// TIA Portal V20 export
// export: Created 2025-12-01T14:56:53.2273381Z, ExportSetting None, DisplayName Totally Integrated Automation Portal, DisplayVersion V20 Update 3, DisplayName TIA Portal Openness, DisplayVersion V20 Update 3, DisplayName TIA Portal Version Control Interface, DisplayVersion V20 Update 3, DisplayName STEP 7 Professional, DisplayVersion V20 Update 3, DisplayName STEP 7 Safety, DisplayVersion V20 Update 2, DisplayName WinCC Basic/Comfort/Advanced, DisplayVersion V20 Update 3, DisplayName WinCC Professional, DisplayVersion V20 Update 3, DisplayName WinCC Unified, DisplayVersion V20 Update 3
FUNCTION_BLOCK "FB368_DesapilCubetas_ERAMAN"   // FB368, LAD
{ S7_Optimized_Access := 'FALSE' }
AUTHOR : PASO
NAME : 20160509
VERSION : 3.8
// stored: AutoNumber false, SetENOAutomatically false
   VAR_INPUT
      Mesa : UInt;   // Mesa de la FB
      Error_Tx : Bool;   // Error en el Tx
      EnTension : Bool;   // Existe Tension en la Mesa
      Termico_Tx : Bool;   // Termico motorrodillo
      PhsMx : Bool;   // Presencia en mesa
      Phs_Pos_Desapil : Bool;   // Posición cilindro medio
      Phs_en_Pinza : Bool;   // Presencia en pinza
      Avance_Tx : Bool;   // Avance del Tx
      CL_UP : Bool;   // Posición cilindro arriba
      CL_DW : Bool;   // Posición cilindro abajo
      EnMovimiento_CL : Bool;
      Gripper_Open : Bool;   // Posición pinza abierta
      Gripper_Close : Bool;   // Posición pinza cerrada
      EnMovimiento_Gripper : Bool;
      TP_UP : Bool;   // Posición tope arriba
      TP_DW : Bool;   // Posición tope abajo
      EnMovimiento_TP : Bool;   // En movimiento el TP1
      MAnt_DescargaAct : Bool;   // E1 >> Mesa Anterior DescargaAct
      AVTF_MAnt_Mx : Bool;
      PTF_Mx_MSig : Bool;
      FTF_Mx_MSig : Bool;
      V_CNT_pHsMx : Int := 1000;   // Valor de Presencia
      V_CNTSeg_pHsMx : Int := 2000;
      V_CNT_ApHsMx : Int := 500;
      V_CNTSeg_ApHsMx : Int := 2000;
      V_CNT_Simultaneo : Int := 2000;   // Valor de Simultaneo
      V_InicioSimultaneo : Int := 0;   // Inicio de Simultaneo. Nota: <= V_CNT_Simultaneo
      V_FinSimultaneo : Int := 0;   // Final de Simultaneo. Nota: <= V_InicioSimultaneo
      V_GripperAbrir : Time := T#200ms;
      V_TOut_Tx_Mx : Int := 10000;   // TimeOut de Entrada por E1
      V_TOut_TP : Int := 2000;   // TimeOut de Tope
      V_TOut_Apil_UPDW : Int := 5000;
      V_TOut_Gripper : Int := 2000;
   END_VAR
   VAR_OUTPUT
      AVTF_Mx_MSig : Bool;
      PTF_MAnt_Mx : Bool;   // E1 >> Mesa Anterior PTF
      FTF_MAnt_Mx : Bool;   // E1 >> Mesa Anterior FTF
      P_Mens_Mx_MSig : Bool;   // S3 >> Mesa Siguiente P_Mens
   END_VAR
   VAR
      Mx_ET00 : Bool;
      Mx_ET01 : Bool;
      Mx_ET02 : Bool;
      Mx_ET08 : Bool;
      Mx_ET09 : Bool;
      Mx_ET10 : Bool;
      Mx_ET11 : Bool;
      Mx_ET12 : Bool;
      Mx_ET50 : Bool;
      Mx_ET51 : Bool;
      Mx_ET501 : Bool;
      Mx_ET502 : Bool;
      Mx_ET503 : Bool;
      Mx_ET504 : Bool;
      Mx_ET505 : Bool;
      Mx_ET506 : Bool;
      STAT_AVTF_Mx_MSig { S7_SetPoint := 'True'} : Bool;
      STAT_FTF_MAnt_Mx : Bool;   // Interna >> FTF de MAnt >> Mx
      MA_Subir_CL : Bool;   // Salida para subir cilindro
      MA_Bajar_CL : Bool;   // Salida para bajar cilindro
      MA_Gripper_Cerrar : Bool;   // Salida cerrar gripper
      MA_Gripper_Abrir : Bool;   // Salida abrir gripper
      En_Movimiento : Bool;
      Simultaneo_Mx : Bool;   // Activo Simultaneo E1
      TMP_Gripper_Cerrar { S7_SetPoint := 'True'} : TON_TIME;
      CNT_pHsMx { S7_SetPoint := 'True'} : "FB910_CNT_UHS";   // CNT de la Presencia
      CNTSeg_pHsMx { S7_SetPoint := 'True'} : "FB910_CNT_UHS";   // CNT de Seguridad de la Presencia
      CNT_ApHsMx { S7_SetPoint := 'True'} : "FB910_CNT_UHS";   // CNT de la Ausencia
      CNTSeg_ApHsMx { S7_SetPoint := 'True'} : "FB910_CNT_UHS";   // CNT de Seguridad de la Ausencia
      CNT_Simultaneo { S7_SetPoint := 'True'} : "FB910_CNT_UHS";   // CNT de Simultaneo
      TMP_EnTension { S7_SetPoint := 'True'} : "FB910_CNT_UHS";
      TOut_Av { S7_SetPoint := 'True'} : "FB910_CNT_UHS";
      TOut_UPDW { S7_SetPoint := 'True'} : "FB910_CNT_UHS";
      TOut_Gripper { S7_SetPoint := 'True'} : "FB910_CNT_UHS";
      TOut_Subir_TP { S7_SetPoint := 'True'} : "FB910_CNT_UHS";
      TOut_Bajar_TP { S7_SetPoint := 'True'} : "FB910_CNT_UHS";
      Manual : "MoviManualMesa_Eraman";
   END_VAR
   VAR_TEMP
      EstadoZona : "EstadoZona";   // Estado de Zona de la Mesa
      EstadoVI : "EstadosMesa_ERAMAN";   // Estado del Vehiculo Inteliguente de la Mesa
      EstadoMaquina : "EstadoMaquina";
      ConfigFB : "UDT_ConfigFB";   // Configuracion de la FB de la Mesa
      Aux_ET00 : Bool;
   END_VAR
BEGIN

REGION Network 1: INICIALIZAR - Recoger las Variables de Estado de la Mesa
   // Se recoge - Estado_CBx
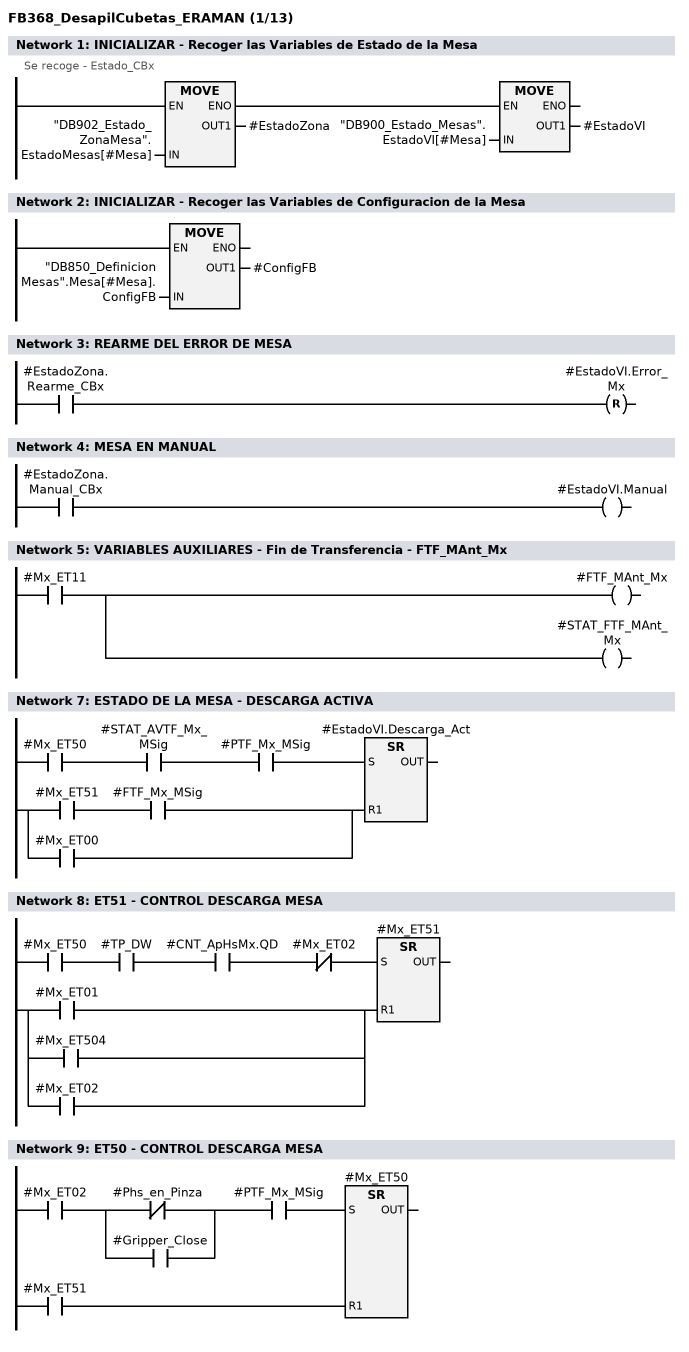
   RUNG wire#powerrail
      Move(in := "DB902_Estado_ZonaMesa".EstadoMesas[#Mesa], out1 => #EstadoZona)
      Move(in := "DB900_Estado_Mesas".EstadoVI[#Mesa], out1 => #EstadoVI)
   END_RUNG
   // the same network as SCL:
   #EstadoZona := "DB902_Estado_ZonaMesa".EstadoMesas[#Mesa];
   #EstadoVI := "DB900_Estado_Mesas".EstadoVI[#Mesa];
END_REGION

REGION Network 2: INICIALIZAR - Recoger las Variables de Configuracion de la Mesa
   RUNG wire#powerrail
      Move(in := "DB850_DefinicionMesas".Mesa[#Mesa].ConfigFB, out1 => #ConfigFB)
   END_RUNG
   // the same network as SCL:
   #ConfigFB := "DB850_DefinicionMesas".Mesa[#Mesa].ConfigFB;
END_REGION

REGION Network 3: REARME DEL ERROR DE MESA
   RUNG wire#powerrail
      Contact( #EstadoZona.Rearme_CBx )
      R_Coil( #EstadoVI.Error_Mx )
   END_RUNG
   // the same network as SCL:
   IF #EstadoZona.Rearme_CBx THEN #EstadoVI.Error_Mx := FALSE; END_IF;
END_REGION

REGION Network 4: MESA EN MANUAL
   RUNG wire#powerrail
      Contact( #EstadoZona.Manual_CBx )
      Coil( #EstadoVI.Manual )
   END_RUNG
   // the same network as SCL:
   #EstadoVI.Manual := #EstadoZona.Manual_CBx;
END_REGION

REGION Network 5: VARIABLES AUXILIARES - Fin de Transferencia - FTF_MAnt_Mx
   RUNG wire#powerrail
      Contact( #Mx_ET11 )
      wire#w1
      Coil( #FTF_MAnt_Mx )
   END_RUNG
   RUNG wire#w1
      Coil( #STAT_FTF_MAnt_Mx )
   END_RUNG
   // the same network as SCL:
   #FTF_MAnt_Mx := #Mx_ET11;
   #STAT_FTF_MAnt_Mx := #Mx_ET11;
END_REGION

REGION Network 6: ----------------------GRAFCET DESCARGA---------------------------
END_REGION

REGION Network 7: ESTADO DE LA MESA - DESCARGA ACTIVA
   RUNG wire#powerrail
      Contact( #Mx_ET50 )
      Contact( #STAT_AVTF_Mx_MSig )
      Contact( #PTF_Mx_MSig )
      S_SR(operand := #EstadoVI.Descarga_Act, r1 := wire#w1)
   END_RUNG
   RUNG wire#powerrail
      Contact( #Mx_ET51 )
      Contact( #FTF_Mx_MSig )
   END_RUNG wire#w1
   RUNG wire#powerrail
      Contact( #Mx_ET00 )
   END_RUNG wire#w1
   // the same network as SCL:
   IF #Mx_ET50 AND #STAT_AVTF_Mx_MSig AND #PTF_Mx_MSig THEN
       #EstadoVI.Descarga_Act := TRUE;   // SR flip-flop
   END_IF;
   IF (#Mx_ET51 AND #FTF_Mx_MSig) OR #Mx_ET00 THEN #EstadoVI.Descarga_Act := FALSE; END_IF;
END_REGION

REGION Network 8: ET51 - CONTROL DESCARGA MESA
   RUNG wire#powerrail
      Contact( #Mx_ET50 )
      Contact( #TP_DW )
      Contact( #CNT_ApHsMx.QD )
      I_Contact( #Mx_ET02 )
      S_SR(operand := #Mx_ET51, r1 := wire#w1)
   END_RUNG
   RUNG wire#powerrail
      Contact( #Mx_ET01 )
   END_RUNG wire#w1
   RUNG wire#powerrail
      Contact( #Mx_ET504 )
   END_RUNG wire#w1
   RUNG wire#powerrail
      Contact( #Mx_ET02 )
   END_RUNG wire#w1
   // the same network as SCL:
   IF #Mx_ET50 AND #TP_DW AND #CNT_ApHsMx.QD AND NOT #Mx_ET02 THEN
       #Mx_ET51 := TRUE;   // SR flip-flop
   END_IF;
   IF #Mx_ET01 OR #Mx_ET504 OR #Mx_ET02 THEN #Mx_ET51 := FALSE; END_IF;
END_REGION

REGION Network 9: ET50 - CONTROL DESCARGA MESA
   RUNG wire#powerrail
      Contact( #Mx_ET02 )
      wire#w1
      I_Contact( #Phs_en_Pinza )
      wire#w2
      Contact( #PTF_Mx_MSig )
      S_SR(operand := #Mx_ET50, r1 := wire#w3)
   END_RUNG
   RUNG wire#w1
      Contact( #Gripper_Close )
   END_RUNG wire#w2
   RUNG wire#powerrail
      Contact( #Mx_ET51 )
   END_RUNG wire#w3
   // the same network as SCL:
   IF #Mx_ET02 AND (NOT #Phs_en_Pinza OR #Gripper_Close) AND #PTF_Mx_MSig THEN
       #Mx_ET50 := TRUE;   // SR flip-flop
   END_IF;
   IF #Mx_ET51 THEN #Mx_ET50 := FALSE; END_IF;
END_REGION

REGION Network 10: ----------------------GRAFCET DESAPILAR--------------------------
END_REGION

REGION Network 11: ET506 >>> Bajar CL
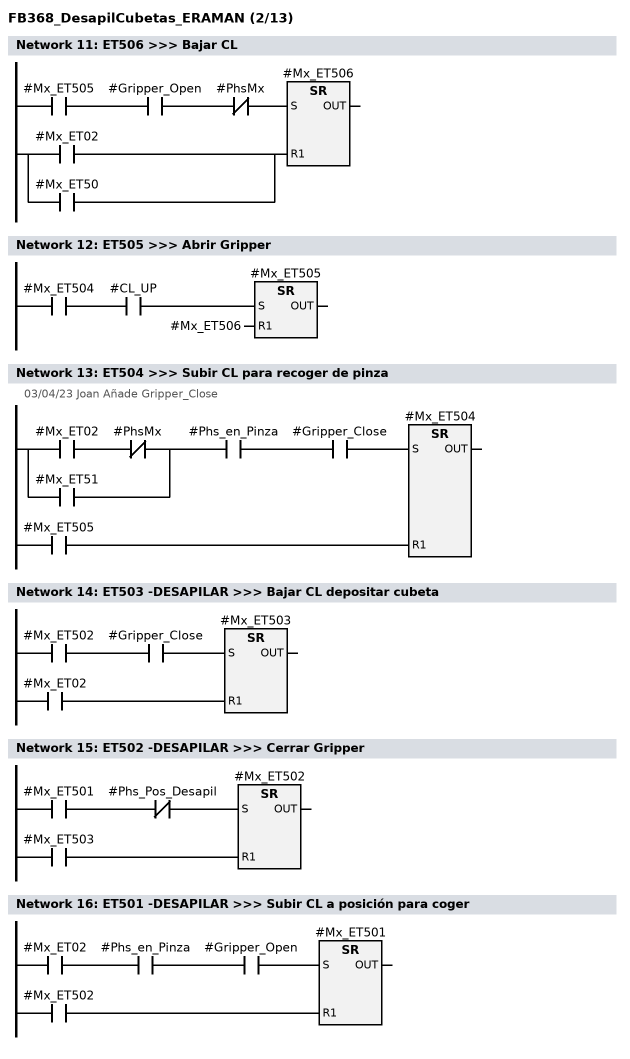
   RUNG wire#powerrail
      Contact( #Mx_ET505 )
      Contact( #Gripper_Open )
      I_Contact( #PhsMx )
      S_SR(operand := #Mx_ET506, r1 := wire#w1)
   END_RUNG
   RUNG wire#powerrail
      Contact( #Mx_ET02 )
   END_RUNG wire#w1
   RUNG wire#powerrail
      Contact( #Mx_ET50 )
   END_RUNG wire#w1
   // the same network as SCL:
   IF #Mx_ET505 AND #Gripper_Open AND NOT #PhsMx THEN
       #Mx_ET506 := TRUE;   // SR flip-flop
   END_IF;
   IF #Mx_ET02 OR #Mx_ET50 THEN #Mx_ET506 := FALSE; END_IF;
END_REGION

REGION Network 12: ET505 >>> Abrir Gripper
   RUNG wire#powerrail
      Contact( #Mx_ET504 )
      Contact( #CL_UP )
      S_SR(operand := #Mx_ET505, r1 := #Mx_ET506)
   END_RUNG
   // the same network as SCL:
   IF #Mx_ET504 AND #CL_UP THEN
       #Mx_ET505 := TRUE;   // SR flip-flop
   END_IF;
   IF #Mx_ET506 THEN #Mx_ET505 := FALSE; END_IF;
END_REGION

REGION Network 13: ET504 >>> Subir CL para recoger de pinza
   // 03/04/23 Joan Añade Gripper_Close
   RUNG wire#powerrail
      Contact( #Mx_ET02 )
      I_Contact( #PhsMx )
      wire#w1
      Contact( #Phs_en_Pinza )
      Contact( #Gripper_Close )
      S_SR(operand := #Mx_ET504, r1 := wire#w2)
   END_RUNG
   RUNG wire#powerrail
      Contact( #Mx_ET51 )
   END_RUNG wire#w1
   RUNG wire#powerrail
      Contact( #Mx_ET505 )
   END_RUNG wire#w2
   // the same network as SCL:
   IF ((#Mx_ET02 AND NOT #PhsMx) OR #Mx_ET51) AND #Phs_en_Pinza AND #Gripper_Close THEN
       #Mx_ET504 := TRUE;   // SR flip-flop
   END_IF;
   IF #Mx_ET505 THEN #Mx_ET504 := FALSE; END_IF;
END_REGION

REGION Network 14: ET503 -DESAPILAR >>> Bajar CL depositar cubeta
   RUNG wire#powerrail
      Contact( #Mx_ET502 )
      Contact( #Gripper_Close )
      S_SR(operand := #Mx_ET503, r1 := wire#w1)
   END_RUNG
   RUNG wire#powerrail
      Contact( #Mx_ET02 )
   END_RUNG wire#w1
   // the same network as SCL:
   IF #Mx_ET502 AND #Gripper_Close THEN
       #Mx_ET503 := TRUE;   // SR flip-flop
   END_IF;
   IF #Mx_ET02 THEN #Mx_ET503 := FALSE; END_IF;
END_REGION

REGION Network 15: ET502 -DESAPILAR >>> Cerrar Gripper
   RUNG wire#powerrail
      Contact( #Mx_ET501 )
      I_Contact( #Phs_Pos_Desapil )
      S_SR(operand := #Mx_ET502, r1 := wire#w1)
   END_RUNG
   RUNG wire#powerrail
      Contact( #Mx_ET503 )
   END_RUNG wire#w1
   // the same network as SCL:
   IF #Mx_ET501 AND NOT #Phs_Pos_Desapil THEN
       #Mx_ET502 := TRUE;   // SR flip-flop
   END_IF;
   IF #Mx_ET503 THEN #Mx_ET502 := FALSE; END_IF;
END_REGION

REGION Network 16: ET501 -DESAPILAR >>> Subir CL a posición para coger
   RUNG wire#powerrail
      Contact( #Mx_ET02 )
      Contact( #Phs_en_Pinza )
      Contact( #Gripper_Open )
      S_SR(operand := #Mx_ET501, r1 := wire#w1)
   END_RUNG
   RUNG wire#powerrail
      Contact( #Mx_ET502 )
   END_RUNG wire#w1
   // the same network as SCL:
   IF #Mx_ET02 AND #Phs_en_Pinza AND #Gripper_Open THEN
       #Mx_ET501 := TRUE;   // SR flip-flop
   END_IF;
   IF #Mx_ET502 THEN #Mx_ET501 := FALSE; END_IF;
END_REGION

REGION Network 17: ET02 -MESA CARGADA >>> Abrir Gripper
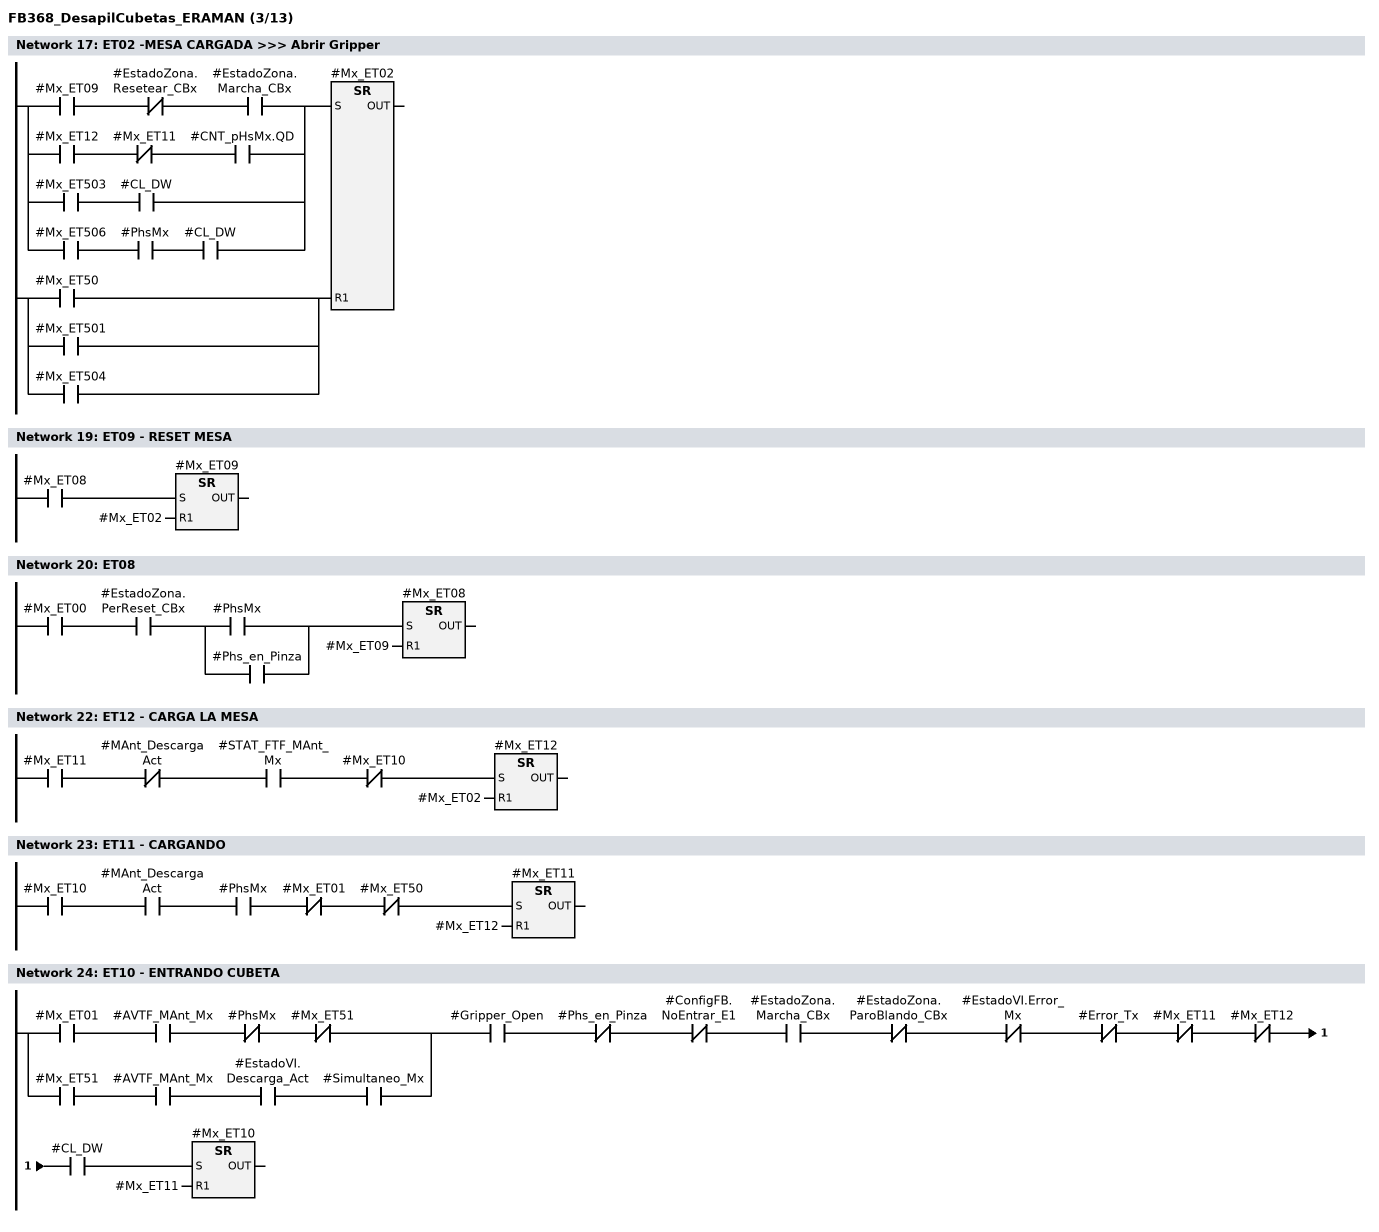
   RUNG wire#powerrail
      Contact( #Mx_ET09 )
      I_Contact( #EstadoZona.Resetear_CBx )
      Contact( #EstadoZona.Marcha_CBx )
      wire#w1
      S_SR(operand := #Mx_ET02, r1 := wire#w2)
   END_RUNG
   RUNG wire#powerrail
      Contact( #Mx_ET12 )
      I_Contact( #Mx_ET11 )
      Contact( #CNT_pHsMx.QD )
   END_RUNG wire#w1
   RUNG wire#powerrail
      Contact( #Mx_ET503 )
      Contact( #CL_DW )
   END_RUNG wire#w1
   RUNG wire#powerrail
      Contact( #Mx_ET506 )
      Contact( #PhsMx )
      Contact( #CL_DW )
   END_RUNG wire#w1
   RUNG wire#powerrail
      Contact( #Mx_ET50 )
   END_RUNG wire#w2
   RUNG wire#powerrail
      Contact( #Mx_ET501 )
   END_RUNG wire#w2
   RUNG wire#powerrail
      Contact( #Mx_ET504 )
   END_RUNG wire#w2
   // the same network as SCL:
   IF (#Mx_ET09 AND NOT #EstadoZona.Resetear_CBx AND #EstadoZona.Marcha_CBx) OR (#Mx_ET12 AND NOT #Mx_ET11 AND #CNT_pHsMx.QD) OR (#Mx_ET503 AND #CL_DW) OR (#Mx_ET506 AND #PhsMx AND #CL_DW) THEN
       #Mx_ET02 := TRUE;   // SR flip-flop
   END_IF;
   IF #Mx_ET50 OR #Mx_ET501 OR #Mx_ET504 THEN #Mx_ET02 := FALSE; END_IF;
END_REGION

REGION Network 18: ----------------------GRAFCET RESET--------------------------
END_REGION

REGION Network 19: ET09 - RESET MESA
   RUNG wire#powerrail
      Contact( #Mx_ET08 )
      S_SR(operand := #Mx_ET09, r1 := #Mx_ET02)
   END_RUNG
   // the same network as SCL:
   IF #Mx_ET08 THEN
       #Mx_ET09 := TRUE;   // SR flip-flop
   END_IF;
   IF #Mx_ET02 THEN #Mx_ET09 := FALSE; END_IF;
END_REGION

REGION Network 20: ET08
   RUNG wire#powerrail
      Contact( #Mx_ET00 )
      Contact( #EstadoZona.PerReset_CBx )
      wire#w1
      Contact( #PhsMx )
      wire#w2
      S_SR(operand := #Mx_ET08, r1 := #Mx_ET09)
   END_RUNG
   RUNG wire#w1
      Contact( #Phs_en_Pinza )
   END_RUNG wire#w2
   // the same network as SCL:
   IF #Mx_ET00 AND #EstadoZona.PerReset_CBx AND (#PhsMx OR #Phs_en_Pinza) THEN
       #Mx_ET08 := TRUE;   // SR flip-flop
   END_IF;
   IF #Mx_ET09 THEN #Mx_ET08 := FALSE; END_IF;
END_REGION

REGION Network 21: ----------------------GRAFCET CARGAR--------------------------
END_REGION

REGION Network 22: ET12 - CARGA LA MESA
   RUNG wire#powerrail
      Contact( #Mx_ET11 )
      I_Contact( #MAnt_DescargaAct )
      Contact( #STAT_FTF_MAnt_Mx )
      I_Contact( #Mx_ET10 )
      S_SR(operand := #Mx_ET12, r1 := #Mx_ET02)
   END_RUNG
   // the same network as SCL:
   IF #Mx_ET11 AND NOT #MAnt_DescargaAct AND #STAT_FTF_MAnt_Mx AND NOT #Mx_ET10 THEN
       #Mx_ET12 := TRUE;   // SR flip-flop
   END_IF;
   IF #Mx_ET02 THEN #Mx_ET12 := FALSE; END_IF;
END_REGION

REGION Network 23: ET11 - CARGANDO
   RUNG wire#powerrail
      Contact( #Mx_ET10 )
      Contact( #MAnt_DescargaAct )
      Contact( #PhsMx )
      I_Contact( #Mx_ET01 )
      I_Contact( #Mx_ET50 )
      S_SR(operand := #Mx_ET11, r1 := #Mx_ET12)
   END_RUNG
   // the same network as SCL:
   IF #Mx_ET10 AND #MAnt_DescargaAct AND #PhsMx AND NOT #Mx_ET01 AND NOT #Mx_ET50 THEN
       #Mx_ET11 := TRUE;   // SR flip-flop
   END_IF;
   IF #Mx_ET12 THEN #Mx_ET11 := FALSE; END_IF;
END_REGION

REGION Network 24: ET10 - ENTRANDO CUBETA
   RUNG wire#powerrail
      Contact( #Mx_ET01 )
      Contact( #AVTF_MAnt_Mx )
      I_Contact( #PhsMx )
      I_Contact( #Mx_ET51 )
      wire#w1
      Contact( #Gripper_Open )
      I_Contact( #Phs_en_Pinza )
      I_Contact( #ConfigFB.NoEntrar_E1 )
      Contact( #EstadoZona.Marcha_CBx )
      I_Contact( #EstadoZona.ParoBlando_CBx )
      I_Contact( #EstadoVI.Error_Mx )
      I_Contact( #Error_Tx )
      I_Contact( #Mx_ET11 )
      I_Contact( #Mx_ET12 )
      Contact( #CL_DW )
      S_SR(operand := #Mx_ET10, r1 := #Mx_ET11)
   END_RUNG
   RUNG wire#powerrail
      Contact( #Mx_ET51 )
      Contact( #AVTF_MAnt_Mx )
      Contact( #EstadoVI.Descarga_Act )
      Contact( #Simultaneo_Mx )
   END_RUNG wire#w1
   // the same network as SCL:
   IF ((#Mx_ET01 AND #AVTF_MAnt_Mx AND NOT #PhsMx AND NOT #Mx_ET51) OR (#Mx_ET51 AND #AVTF_MAnt_Mx AND #EstadoVI.Descarga_Act AND #Simultaneo_Mx)) AND #Gripper_Open AND NOT #Phs_en_Pinza AND NOT #ConfigFB.NoEntrar_E1 AND #EstadoZona.Marcha_CBx AND NOT #EstadoZona.ParoBlando_CBx AND NOT #EstadoVI.Error_Mx AND NOT #Error_Tx AND NOT #Mx_ET11 AND NOT #Mx_ET12 AND #CL_DW THEN
       #Mx_ET10 := TRUE;   // SR flip-flop
   END_IF;
   IF #Mx_ET11 THEN #Mx_ET10 := FALSE; END_IF;
END_REGION

REGION Network 25: ----------------------GRAFCET REPOSO/VACIO--------------------------
END_REGION

REGION Network 26: ET01 - ESTADO REPOSO VACIO
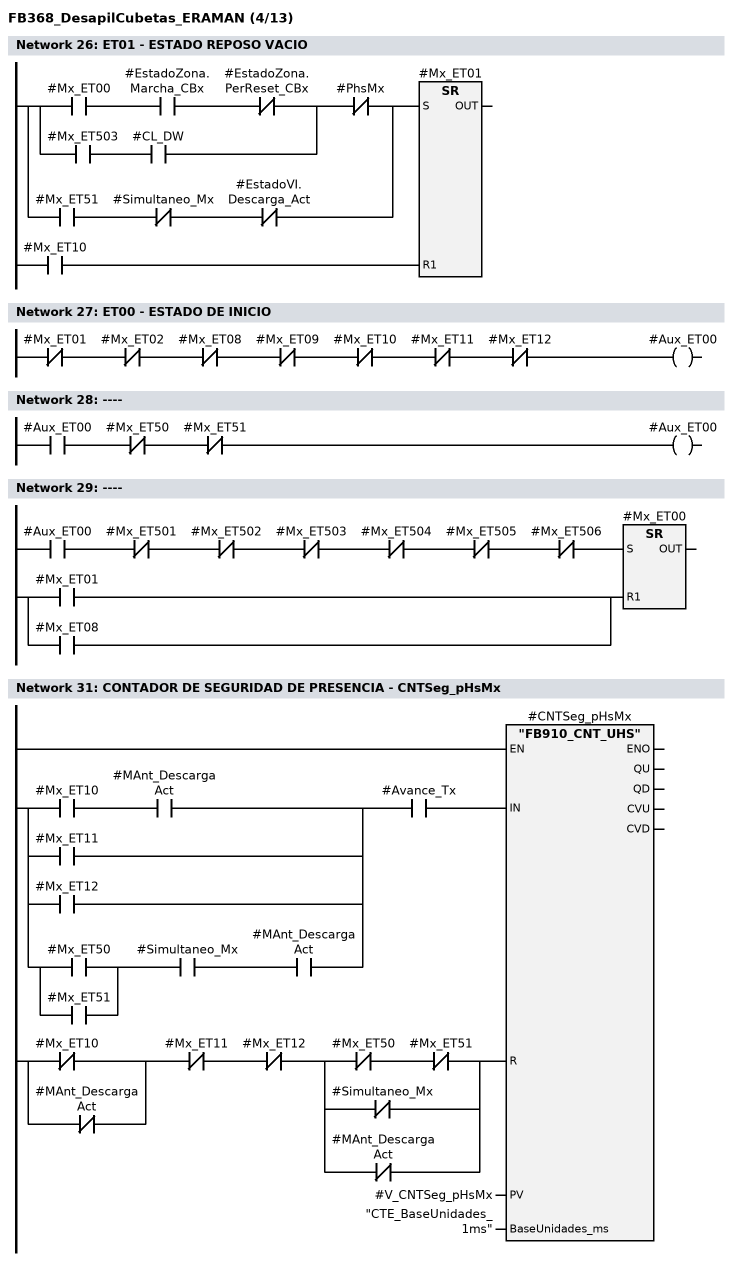
   RUNG wire#powerrail
      Contact( #Mx_ET00 )
      Contact( #EstadoZona.Marcha_CBx )
      I_Contact( #EstadoZona.PerReset_CBx )
      wire#w1
      I_Contact( #PhsMx )
      wire#w2
      S_SR(operand := #Mx_ET01, r1 := wire#w3)
   END_RUNG
   RUNG wire#powerrail
      Contact( #Mx_ET503 )
      Contact( #CL_DW )
   END_RUNG wire#w1
   RUNG wire#powerrail
      Contact( #Mx_ET51 )
      I_Contact( #Simultaneo_Mx )
      I_Contact( #EstadoVI.Descarga_Act )
   END_RUNG wire#w2
   RUNG wire#powerrail
      Contact( #Mx_ET10 )
   END_RUNG wire#w3
   // the same network as SCL:
   IF (((#Mx_ET00 AND #EstadoZona.Marcha_CBx AND NOT #EstadoZona.PerReset_CBx) OR (#Mx_ET503 AND #CL_DW)) AND NOT #PhsMx) OR (#Mx_ET51 AND NOT #Simultaneo_Mx AND NOT #EstadoVI.Descarga_Act) THEN
       #Mx_ET01 := TRUE;   // SR flip-flop
   END_IF;
   IF #Mx_ET10 THEN #Mx_ET01 := FALSE; END_IF;
END_REGION

REGION Network 27: ET00 - ESTADO DE INICIO
   RUNG wire#powerrail
      I_Contact( #Mx_ET01 )
      I_Contact( #Mx_ET02 )
      I_Contact( #Mx_ET08 )
      I_Contact( #Mx_ET09 )
      I_Contact( #Mx_ET10 )
      I_Contact( #Mx_ET11 )
      I_Contact( #Mx_ET12 )
      Coil( #Aux_ET00 )
   END_RUNG
   // the same network as SCL:
   #Aux_ET00 := NOT #Mx_ET01 AND NOT #Mx_ET02 AND NOT #Mx_ET08 AND NOT #Mx_ET09 AND NOT #Mx_ET10 AND NOT #Mx_ET11 AND NOT #Mx_ET12;
END_REGION

REGION Network 28: ----
   RUNG wire#powerrail
      Contact( #Aux_ET00 )
      I_Contact( #Mx_ET50 )
      I_Contact( #Mx_ET51 )
      Coil( #Aux_ET00 )
   END_RUNG
   // the same network as SCL:
   #Aux_ET00 := #Aux_ET00 AND NOT #Mx_ET50 AND NOT #Mx_ET51;
END_REGION

REGION Network 29: ----
   RUNG wire#powerrail
      Contact( #Aux_ET00 )
      I_Contact( #Mx_ET501 )
      I_Contact( #Mx_ET502 )
      I_Contact( #Mx_ET503 )
      I_Contact( #Mx_ET504 )
      I_Contact( #Mx_ET505 )
      I_Contact( #Mx_ET506 )
      S_SR(operand := #Mx_ET00, r1 := wire#w1)
   END_RUNG
   RUNG wire#powerrail
      Contact( #Mx_ET01 )
   END_RUNG wire#w1
   RUNG wire#powerrail
      Contact( #Mx_ET08 )
   END_RUNG wire#w1
   // the same network as SCL:
   IF #Aux_ET00 AND NOT #Mx_ET501 AND NOT #Mx_ET502 AND NOT #Mx_ET503 AND NOT #Mx_ET504 AND NOT #Mx_ET505 AND NOT #Mx_ET506 THEN
       #Mx_ET00 := TRUE;   // SR flip-flop
   END_IF;
   IF #Mx_ET01 OR #Mx_ET08 THEN #Mx_ET00 := FALSE; END_IF;
END_REGION

REGION Network 30: ----------------------TEMPORIZADORES / CONTADORES -------------------------
END_REGION

REGION Network 31: CONTADOR DE SEGURIDAD DE PRESENCIA - CNTSeg_pHsMx
   RUNG wire#powerrail
      #CNTSeg_pHsMx(IN := wire#w3, R := wire#w6, PV := #V_CNTSeg_pHsMx, BaseUnidades_ms := "CTE_BaseUnidades_1ms", QU =>, QD =>, CVU =>, CVD =>)
   END_RUNG
   RUNG wire#powerrail
      Contact( #Mx_ET10 )
      Contact( #MAnt_DescargaAct )
      wire#w1
      Contact( #Avance_Tx )
   END_RUNG wire#w3
   RUNG wire#powerrail
      Contact( #Mx_ET11 )
   END_RUNG wire#w1
   RUNG wire#powerrail
      Contact( #Mx_ET12 )
   END_RUNG wire#w1
   RUNG wire#powerrail
      Contact( #Mx_ET50 )
      wire#w2
      Contact( #Simultaneo_Mx )
      Contact( #MAnt_DescargaAct )
   END_RUNG wire#w1
   RUNG wire#powerrail
      Contact( #Mx_ET51 )
   END_RUNG wire#w2
   RUNG wire#powerrail
      I_Contact( #Mx_ET10 )
      wire#w4
      I_Contact( #Mx_ET11 )
      I_Contact( #Mx_ET12 )
      wire#w5
      I_Contact( #Mx_ET50 )
      I_Contact( #Mx_ET51 )
   END_RUNG wire#w6
   RUNG wire#powerrail
      I_Contact( #MAnt_DescargaAct )
   END_RUNG wire#w4
   RUNG wire#w5
      I_Contact( #Simultaneo_Mx )
   END_RUNG wire#w6
   RUNG wire#w5
      I_Contact( #MAnt_DescargaAct )
   END_RUNG wire#w6
   // the same network as SCL:
   #CNTSeg_pHsMx(IN := ((#Mx_ET10 AND #MAnt_DescargaAct) OR #Mx_ET11 OR #Mx_ET12 OR ((#Mx_ET50 OR #Mx_ET51) AND #Simultaneo_Mx AND #MAnt_DescargaAct)) AND #Avance_Tx,   // "FB910_CNT_UHS"
                 R := (NOT #Mx_ET10 OR NOT #MAnt_DescargaAct) AND NOT #Mx_ET11 AND NOT #Mx_ET12 AND ((NOT #Mx_ET50 AND NOT #Mx_ET51) OR NOT #Simultaneo_Mx OR NOT #MAnt_DescargaAct),
                 PV := #V_CNTSeg_pHsMx,
                 BaseUnidades_ms := "CTE_BaseUnidades_1ms");
END_REGION

REGION Network 32: CONTADOR DE PRESENCIA - CNT_pHsMx
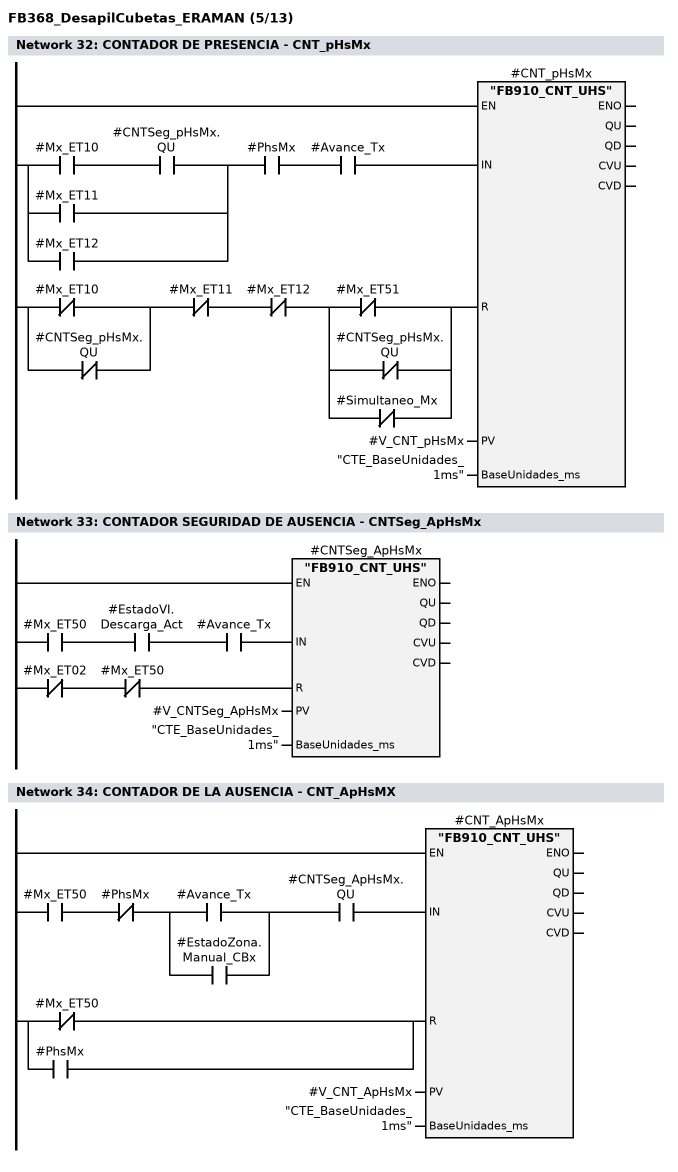
   RUNG wire#powerrail
      #CNT_pHsMx(IN := wire#w2, R := wire#w5, PV := #V_CNT_pHsMx, BaseUnidades_ms := "CTE_BaseUnidades_1ms", QU =>, QD =>, CVU =>, CVD =>)
   END_RUNG
   RUNG wire#powerrail
      Contact( #Mx_ET10 )
      Contact( #CNTSeg_pHsMx.QU )
      wire#w1
      Contact( #PhsMx )
      Contact( #Avance_Tx )
   END_RUNG wire#w2
   RUNG wire#powerrail
      Contact( #Mx_ET11 )
   END_RUNG wire#w1
   RUNG wire#powerrail
      Contact( #Mx_ET12 )
   END_RUNG wire#w1
   RUNG wire#powerrail
      I_Contact( #Mx_ET10 )
      wire#w3
      I_Contact( #Mx_ET11 )
      I_Contact( #Mx_ET12 )
      wire#w4
      I_Contact( #Mx_ET51 )
   END_RUNG wire#w5
   RUNG wire#powerrail
      I_Contact( #CNTSeg_pHsMx.QU )
   END_RUNG wire#w3
   RUNG wire#w4
      I_Contact( #CNTSeg_pHsMx.QU )
   END_RUNG wire#w5
   RUNG wire#w4
      I_Contact( #Simultaneo_Mx )
   END_RUNG wire#w5
   // the same network as SCL:
   #CNT_pHsMx(IN := ((#Mx_ET10 AND #CNTSeg_pHsMx.QU) OR #Mx_ET11 OR #Mx_ET12) AND #PhsMx AND #Avance_Tx,   // "FB910_CNT_UHS"
              R := (NOT #Mx_ET10 OR NOT #CNTSeg_pHsMx.QU) AND NOT #Mx_ET11 AND NOT #Mx_ET12 AND (NOT #Mx_ET51 OR NOT #CNTSeg_pHsMx.QU OR NOT #Simultaneo_Mx),
              PV := #V_CNT_pHsMx,
              BaseUnidades_ms := "CTE_BaseUnidades_1ms");
END_REGION

REGION Network 33: CONTADOR SEGURIDAD DE AUSENCIA - CNTSeg_ApHsMx
   RUNG wire#powerrail
      #CNTSeg_ApHsMx(IN := wire#w1, R := wire#w2, PV := #V_CNTSeg_ApHsMx, BaseUnidades_ms := "CTE_BaseUnidades_1ms", QU =>, QD =>, CVU =>, CVD =>)
   END_RUNG
   RUNG wire#powerrail
      Contact( #Mx_ET50 )
      Contact( #EstadoVI.Descarga_Act )
      Contact( #Avance_Tx )
   END_RUNG wire#w1
   RUNG wire#powerrail
      I_Contact( #Mx_ET02 )
      I_Contact( #Mx_ET50 )
   END_RUNG wire#w2
   // the same network as SCL:
   #CNTSeg_ApHsMx(IN := #Mx_ET50 AND #EstadoVI.Descarga_Act AND #Avance_Tx,   // "FB910_CNT_UHS"
                  R := NOT #Mx_ET02 AND NOT #Mx_ET50,
                  PV := #V_CNTSeg_ApHsMx,
                  BaseUnidades_ms := "CTE_BaseUnidades_1ms");
END_REGION

REGION Network 34: CONTADOR DE LA AUSENCIA - CNT_ApHsMX
   RUNG wire#powerrail
      #CNT_ApHsMx(IN := wire#w3, R := wire#w4, PV := #V_CNT_ApHsMx, BaseUnidades_ms := "CTE_BaseUnidades_1ms", QU =>, QD =>, CVU =>, CVD =>)
   END_RUNG
   RUNG wire#powerrail
      Contact( #Mx_ET50 )
      I_Contact( #PhsMx )
      wire#w1
      Contact( #Avance_Tx )
      wire#w2
      Contact( #CNTSeg_ApHsMx.QU )
   END_RUNG wire#w3
   RUNG wire#w1
      Contact( #EstadoZona.Manual_CBx )
   END_RUNG wire#w2
   RUNG wire#powerrail
      I_Contact( #Mx_ET50 )
   END_RUNG wire#w4
   RUNG wire#powerrail
      Contact( #PhsMx )
   END_RUNG wire#w4
   // the same network as SCL:
   #CNT_ApHsMx(IN := #Mx_ET50 AND NOT #PhsMx AND (#Avance_Tx OR #EstadoZona.Manual_CBx) AND #CNTSeg_ApHsMx.QU,   // "FB910_CNT_UHS"
               R := NOT #Mx_ET50 OR #PhsMx,
               PV := #V_CNT_ApHsMx,
               BaseUnidades_ms := "CTE_BaseUnidades_1ms");
END_REGION

REGION Network 35: CONTADOR DE SIMULTANEO
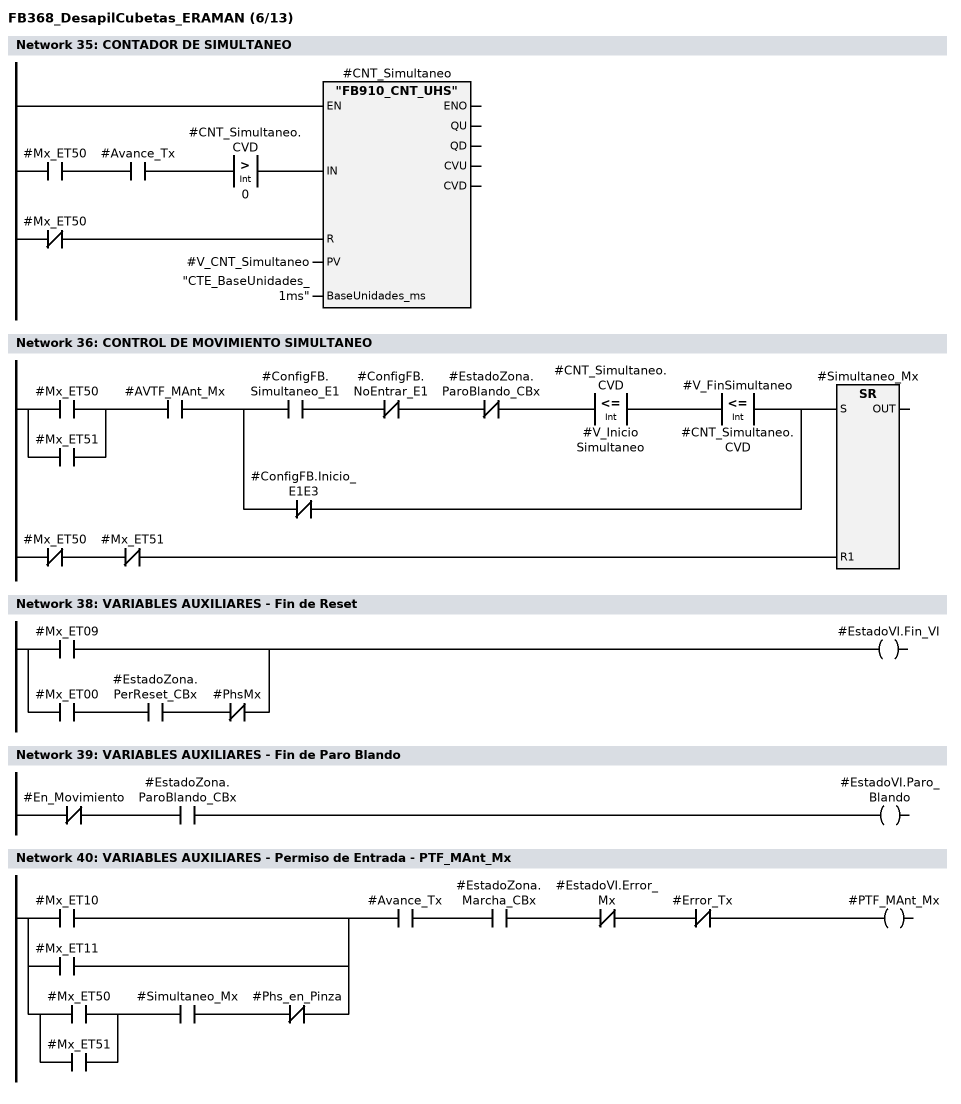
   RUNG wire#powerrail
      #CNT_Simultaneo(IN := wire#w1, R := wire#w2, PV := #V_CNT_Simultaneo, BaseUnidades_ms := "CTE_BaseUnidades_1ms", QU =>, QD =>, CVU =>, CVD =>)
   END_RUNG
   RUNG wire#powerrail
      Contact( #Mx_ET50 )
      Contact( #Avance_Tx )
      { S7_Templates := "SrcType := Int" } GT_Contact(in1 := #CNT_Simultaneo.CVD, in2 := 0)
   END_RUNG wire#w1
   RUNG wire#powerrail
      I_Contact( #Mx_ET50 )
   END_RUNG wire#w2
   // the same network as SCL:
   #CNT_Simultaneo(IN := #Mx_ET50 AND #Avance_Tx AND (#CNT_Simultaneo.CVD > 0),   // "FB910_CNT_UHS"
                   R := NOT #Mx_ET50,
                   PV := #V_CNT_Simultaneo,
                   BaseUnidades_ms := "CTE_BaseUnidades_1ms");
END_REGION

REGION Network 36: CONTROL DE MOVIMIENTO SIMULTANEO
   RUNG wire#powerrail
      Contact( #Mx_ET50 )
      wire#w1
      Contact( #AVTF_MAnt_Mx )
      wire#w2
      Contact( #ConfigFB.Simultaneo_E1 )
      I_Contact( #ConfigFB.NoEntrar_E1 )
      I_Contact( #EstadoZona.ParoBlando_CBx )
      { S7_Templates := "SrcType := Int" } LE_Contact(in1 := #CNT_Simultaneo.CVD, in2 := #V_InicioSimultaneo)
      { S7_Templates := "SrcType := Int" } LE_Contact(in1 := #V_FinSimultaneo, in2 := #CNT_Simultaneo.CVD)
      wire#w3
      S_SR(operand := #Simultaneo_Mx, r1 := wire#w4)
   END_RUNG
   RUNG wire#powerrail
      Contact( #Mx_ET51 )
   END_RUNG wire#w1
   RUNG wire#w2
      I_Contact( #ConfigFB.Inicio_E1E3 )
   END_RUNG wire#w3
   RUNG wire#powerrail
      I_Contact( #Mx_ET50 )
      I_Contact( #Mx_ET51 )
   END_RUNG wire#w4
   // the same network as SCL:
   IF (#Mx_ET50 OR #Mx_ET51) AND #AVTF_MAnt_Mx AND ((#ConfigFB.Simultaneo_E1 AND NOT #ConfigFB.NoEntrar_E1 AND NOT #EstadoZona.ParoBlando_CBx AND (#CNT_Simultaneo.CVD <= #V_InicioSimultaneo) AND (#V_FinSimultaneo <= #CNT_Simultaneo.CVD)) OR NOT #ConfigFB.Inicio_E1E3) THEN
       #Simultaneo_Mx := TRUE;   // SR flip-flop
   END_IF;
   IF NOT #Mx_ET50 AND NOT #Mx_ET51 THEN #Simultaneo_Mx := FALSE; END_IF;
END_REGION

REGION Network 37: ----------------------VARIABLES AUXILIARES -------------------------
END_REGION

REGION Network 38: VARIABLES AUXILIARES - Fin de Reset
   RUNG wire#powerrail
      Contact( #Mx_ET09 )
      wire#w1
      Coil( #EstadoVI.Fin_VI )
   END_RUNG
   RUNG wire#powerrail
      Contact( #Mx_ET00 )
      Contact( #EstadoZona.PerReset_CBx )
      I_Contact( #PhsMx )
   END_RUNG wire#w1
   // the same network as SCL:
   #EstadoVI.Fin_VI := #Mx_ET09 OR (#Mx_ET00 AND #EstadoZona.PerReset_CBx AND NOT #PhsMx);
END_REGION

REGION Network 39: VARIABLES AUXILIARES - Fin de Paro Blando
   RUNG wire#powerrail
      I_Contact( #En_Movimiento )
      Contact( #EstadoZona.ParoBlando_CBx )
      Coil( #EstadoVI.Paro_Blando )
   END_RUNG
   // the same network as SCL:
   #EstadoVI.Paro_Blando := NOT #En_Movimiento AND #EstadoZona.ParoBlando_CBx;
END_REGION

REGION Network 40: VARIABLES AUXILIARES - Permiso de Entrada - PTF_MAnt_Mx
   RUNG wire#powerrail
      Contact( #Mx_ET10 )
      wire#w1
      Contact( #Avance_Tx )
      Contact( #EstadoZona.Marcha_CBx )
      I_Contact( #EstadoVI.Error_Mx )
      I_Contact( #Error_Tx )
      Coil( #PTF_MAnt_Mx )
   END_RUNG
   RUNG wire#powerrail
      Contact( #Mx_ET11 )
   END_RUNG wire#w1
   RUNG wire#powerrail
      Contact( #Mx_ET50 )
      wire#w2
      Contact( #Simultaneo_Mx )
      I_Contact( #Phs_en_Pinza )
   END_RUNG wire#w1
   RUNG wire#powerrail
      Contact( #Mx_ET51 )
   END_RUNG wire#w2
   // the same network as SCL:
   #PTF_MAnt_Mx := (#Mx_ET10 OR #Mx_ET11 OR ((#Mx_ET50 OR #Mx_ET51) AND #Simultaneo_Mx AND NOT #Phs_en_Pinza)) AND #Avance_Tx AND #EstadoZona.Marcha_CBx AND NOT #EstadoVI.Error_Mx AND NOT #Error_Tx;
END_REGION

REGION Network 41: VARIABLES AUXILIARES - Aviso de Salida - AVTF_Mx_MSig
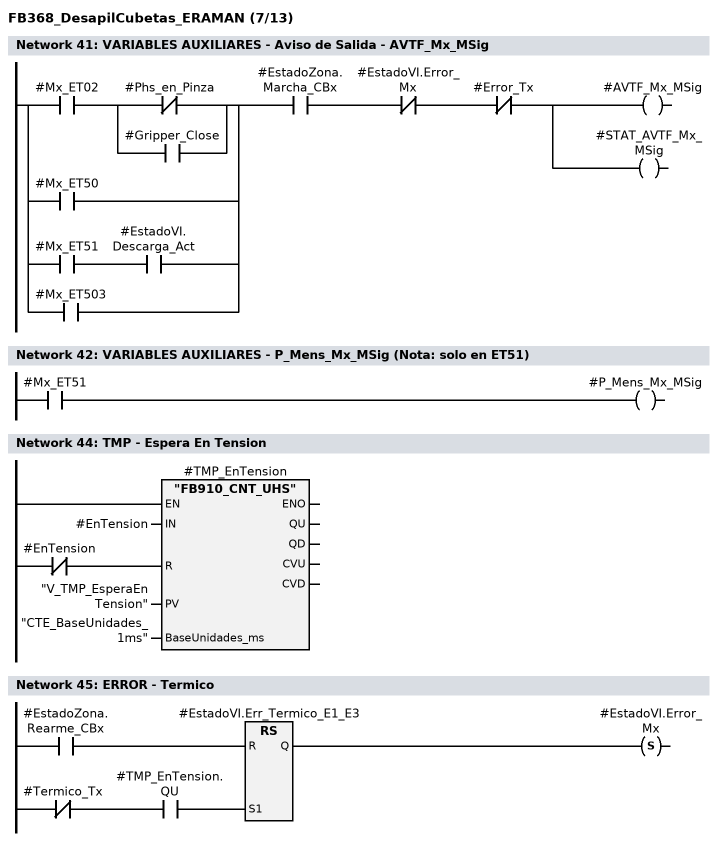
   RUNG wire#powerrail
      Contact( #Mx_ET02 )
      wire#w1
      I_Contact( #Phs_en_Pinza )
      wire#w2
      Contact( #EstadoZona.Marcha_CBx )
      I_Contact( #EstadoVI.Error_Mx )
      I_Contact( #Error_Tx )
      wire#w3
      Coil( #AVTF_Mx_MSig )
   END_RUNG
   RUNG wire#w1
      Contact( #Gripper_Close )
   END_RUNG wire#w2
   RUNG wire#powerrail
      Contact( #Mx_ET50 )
   END_RUNG wire#w2
   RUNG wire#powerrail
      Contact( #Mx_ET51 )
      Contact( #EstadoVI.Descarga_Act )
   END_RUNG wire#w2
   RUNG wire#powerrail
      Contact( #Mx_ET503 )
   END_RUNG wire#w2
   RUNG wire#w3
      Coil( #STAT_AVTF_Mx_MSig )
   END_RUNG
   // the same network as SCL:
   #AVTF_Mx_MSig := ((#Mx_ET02 AND (NOT #Phs_en_Pinza OR #Gripper_Close)) OR #Mx_ET50 OR (#Mx_ET51 AND #EstadoVI.Descarga_Act) OR #Mx_ET503) AND #EstadoZona.Marcha_CBx AND NOT #EstadoVI.Error_Mx AND NOT #Error_Tx;
   #STAT_AVTF_Mx_MSig := #AVTF_Mx_MSig;
END_REGION

REGION Network 42: VARIABLES AUXILIARES - P_Mens_Mx_MSig (Nota: solo en ET51)
   RUNG wire#powerrail
      Contact( #Mx_ET51 )
      Coil( #P_Mens_Mx_MSig )
   END_RUNG
   // the same network as SCL:
   #P_Mens_Mx_MSig := #Mx_ET51;
END_REGION

REGION Network 43: ----------------------ERRORES -------------------------
END_REGION

REGION Network 44: TMP - Espera En Tension
   RUNG wire#powerrail
      #TMP_EnTension(R := wire#w1, IN := #EnTension, PV := "V_TMP_EsperaEnTension", BaseUnidades_ms := "CTE_BaseUnidades_1ms", QU =>, QD =>, CVU =>, CVD =>)
   END_RUNG
   RUNG wire#powerrail
      I_Contact( #EnTension )
   END_RUNG wire#w1
   // the same network as SCL:
   #TMP_EnTension(IN := #EnTension,   // "FB910_CNT_UHS"
                  R := NOT #EnTension,
                  PV := "V_TMP_EsperaEnTension",
                  BaseUnidades_ms := "CTE_BaseUnidades_1ms");
END_REGION

REGION Network 45: ERROR - Termico
   RUNG wire#powerrail
      Contact( #EstadoZona.Rearme_CBx )
      S_RS(operand := #EstadoVI.Err_Termico_E1_E3, s1 := wire#w1)
      S_Coil( #EstadoVI.Error_Mx )
   END_RUNG
   RUNG wire#powerrail
      I_Contact( #Termico_Tx )
      Contact( #TMP_EnTension.QU )
   END_RUNG wire#w1
   // the same network as SCL:
   IF #EstadoZona.Rearme_CBx THEN
       #EstadoVI.Err_Termico_E1_E3 := FALSE;   // RS flip-flop
   END_IF;
   IF NOT #Termico_Tx AND #TMP_EnTension.QU THEN #EstadoVI.Err_Termico_E1_E3 := TRUE; END_IF;
   IF #EstadoVI.Err_Termico_E1_E3 THEN #EstadoVI.Error_Mx := TRUE; END_IF;
END_REGION

REGION Network 46: TMP - ERROR - TimeOut Avance
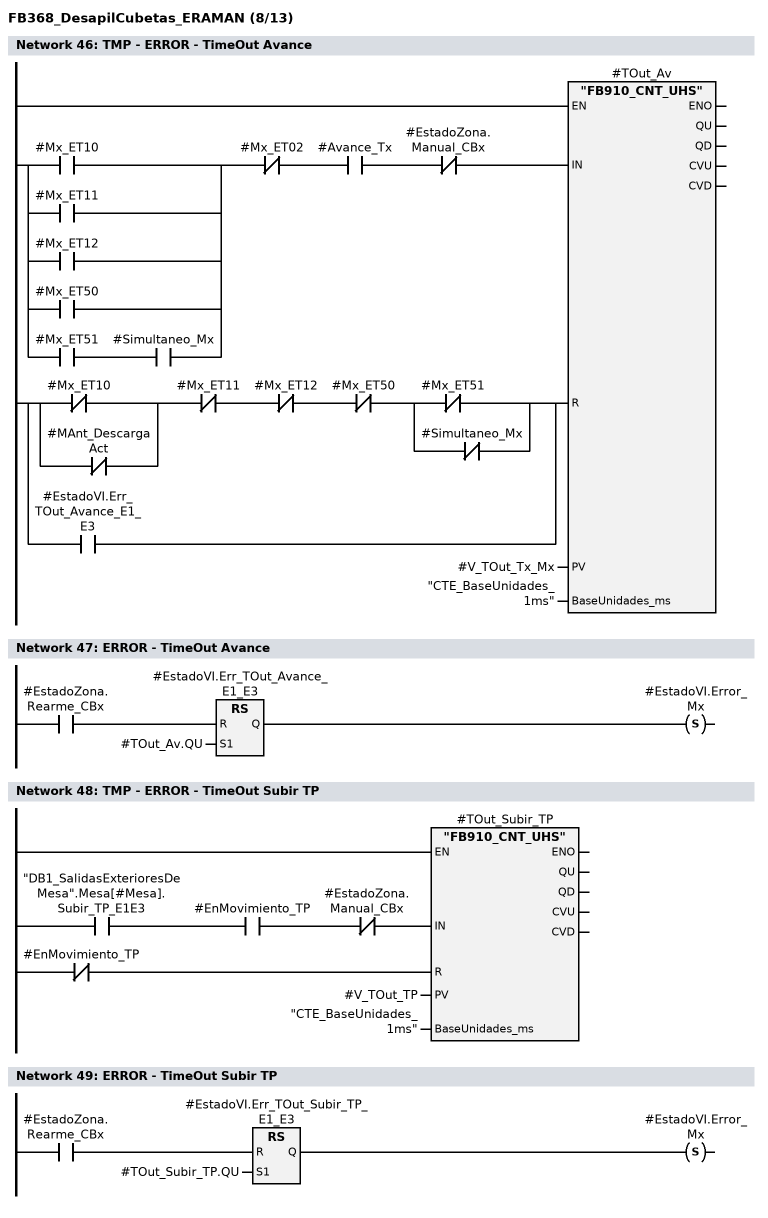
   RUNG wire#powerrail
      #TOut_Av(IN := wire#w2, R := wire#w5, PV := #V_TOut_Tx_Mx, BaseUnidades_ms := "CTE_BaseUnidades_1ms", QU =>, QD =>, CVU =>, CVD =>)
   END_RUNG
   RUNG wire#powerrail
      Contact( #Mx_ET10 )
      wire#w1
      I_Contact( #Mx_ET02 )
      Contact( #Avance_Tx )
      I_Contact( #EstadoZona.Manual_CBx )
   END_RUNG wire#w2
   RUNG wire#powerrail
      Contact( #Mx_ET11 )
   END_RUNG wire#w1
   RUNG wire#powerrail
      Contact( #Mx_ET12 )
   END_RUNG wire#w1
   RUNG wire#powerrail
      Contact( #Mx_ET50 )
   END_RUNG wire#w1
   RUNG wire#powerrail
      Contact( #Mx_ET51 )
      Contact( #Simultaneo_Mx )
   END_RUNG wire#w1
   RUNG wire#powerrail
      I_Contact( #Mx_ET10 )
      wire#w3
      I_Contact( #Mx_ET11 )
      I_Contact( #Mx_ET12 )
      I_Contact( #Mx_ET50 )
      wire#w4
      I_Contact( #Mx_ET51 )
   END_RUNG wire#w5
   RUNG wire#powerrail
      I_Contact( #MAnt_DescargaAct )
   END_RUNG wire#w3
   RUNG wire#w4
      I_Contact( #Simultaneo_Mx )
   END_RUNG wire#w5
   RUNG wire#powerrail
      Contact( #EstadoVI.Err_TOut_Avance_E1_E3 )
   END_RUNG wire#w5
   // the same network as SCL:
   #TOut_Av(IN := (#Mx_ET10 OR #Mx_ET11 OR #Mx_ET12 OR #Mx_ET50 OR (#Mx_ET51 AND #Simultaneo_Mx)) AND NOT #Mx_ET02 AND #Avance_Tx AND NOT #EstadoZona.Manual_CBx,   // "FB910_CNT_UHS"
            R := ((NOT #Mx_ET10 OR NOT #MAnt_DescargaAct) AND NOT #Mx_ET11 AND NOT #Mx_ET12 AND NOT #Mx_ET50 AND (NOT #Mx_ET51 OR NOT #Simultaneo_Mx)) OR #EstadoVI.Err_TOut_Avance_E1_E3,
            PV := #V_TOut_Tx_Mx,
            BaseUnidades_ms := "CTE_BaseUnidades_1ms");
END_REGION

REGION Network 47: ERROR - TimeOut Avance
   RUNG wire#powerrail
      Contact( #EstadoZona.Rearme_CBx )
      S_RS(operand := #EstadoVI.Err_TOut_Avance_E1_E3, s1 := #TOut_Av.QU)
      S_Coil( #EstadoVI.Error_Mx )
   END_RUNG
   // the same network as SCL:
   IF #EstadoZona.Rearme_CBx THEN
       #EstadoVI.Err_TOut_Avance_E1_E3 := FALSE;   // RS flip-flop
   END_IF;
   IF #TOut_Av.QU THEN #EstadoVI.Err_TOut_Avance_E1_E3 := TRUE; END_IF;
   IF #EstadoVI.Err_TOut_Avance_E1_E3 THEN #EstadoVI.Error_Mx := TRUE; END_IF;
END_REGION

REGION Network 48: TMP - ERROR - TimeOut Subir TP
   RUNG wire#powerrail
      #TOut_Subir_TP(IN := wire#w1, R := wire#w2, PV := #V_TOut_TP, BaseUnidades_ms := "CTE_BaseUnidades_1ms", QU =>, QD =>, CVU =>, CVD =>)
   END_RUNG
   RUNG wire#powerrail
      Contact( "DB1_SalidasExterioresDeMesa".Mesa[#Mesa].Subir_TP_E1E3 )
      Contact( #EnMovimiento_TP )
      I_Contact( #EstadoZona.Manual_CBx )
   END_RUNG wire#w1
   RUNG wire#powerrail
      I_Contact( #EnMovimiento_TP )
   END_RUNG wire#w2
   // the same network as SCL:
   #TOut_Subir_TP(IN := "DB1_SalidasExterioresDeMesa".Mesa[#Mesa].Subir_TP_E1E3 AND #EnMovimiento_TP AND NOT #EstadoZona.Manual_CBx,   // "FB910_CNT_UHS"
                  R := NOT #EnMovimiento_TP,
                  PV := #V_TOut_TP,
                  BaseUnidades_ms := "CTE_BaseUnidades_1ms");
END_REGION

REGION Network 49: ERROR - TimeOut Subir TP
   RUNG wire#powerrail
      Contact( #EstadoZona.Rearme_CBx )
      S_RS(operand := #EstadoVI.Err_TOut_Subir_TP_E1_E3, s1 := #TOut_Subir_TP.QU)
      S_Coil( #EstadoVI.Error_Mx )
   END_RUNG
   // the same network as SCL:
   IF #EstadoZona.Rearme_CBx THEN
       #EstadoVI.Err_TOut_Subir_TP_E1_E3 := FALSE;   // RS flip-flop
   END_IF;
   IF #TOut_Subir_TP.QU THEN #EstadoVI.Err_TOut_Subir_TP_E1_E3 := TRUE; END_IF;
   IF #EstadoVI.Err_TOut_Subir_TP_E1_E3 THEN #EstadoVI.Error_Mx := TRUE; END_IF;
END_REGION

REGION Network 50: TMP - ERROR - TimeOut Bajar TP
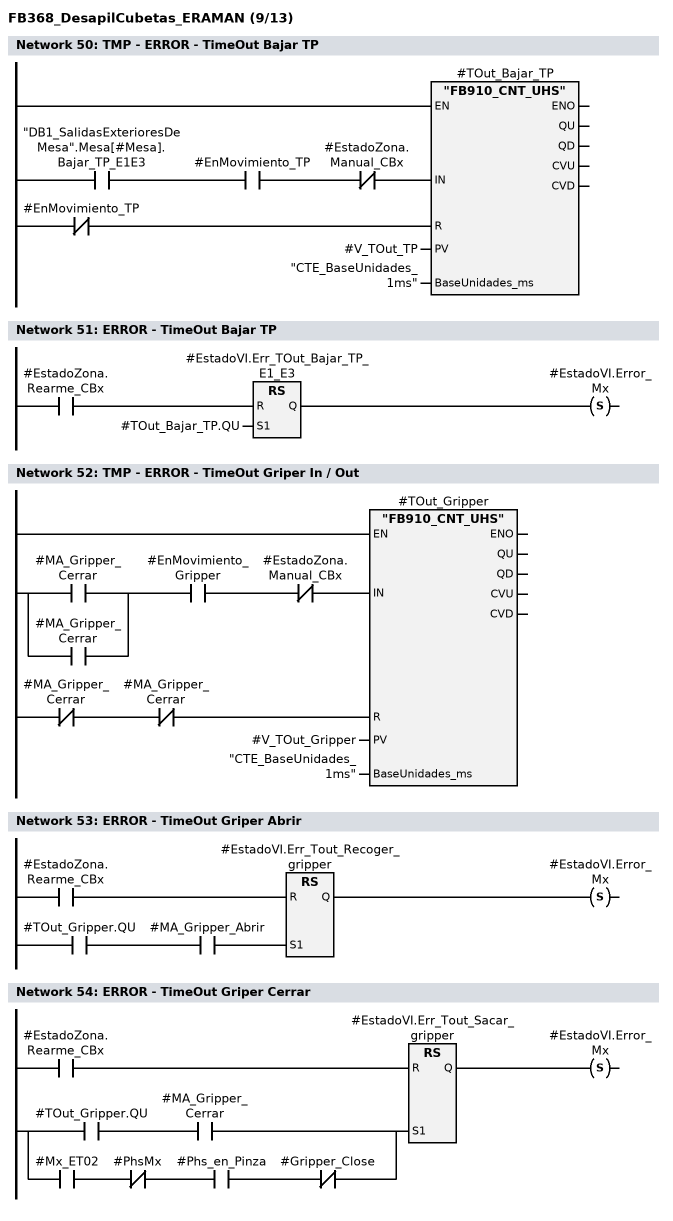
   RUNG wire#powerrail
      #TOut_Bajar_TP(IN := wire#w1, R := wire#w2, PV := #V_TOut_TP, BaseUnidades_ms := "CTE_BaseUnidades_1ms", QU =>, QD =>, CVU =>, CVD =>)
   END_RUNG
   RUNG wire#powerrail
      Contact( "DB1_SalidasExterioresDeMesa".Mesa[#Mesa].Bajar_TP_E1E3 )
      Contact( #EnMovimiento_TP )
      I_Contact( #EstadoZona.Manual_CBx )
   END_RUNG wire#w1
   RUNG wire#powerrail
      I_Contact( #EnMovimiento_TP )
   END_RUNG wire#w2
   // the same network as SCL:
   #TOut_Bajar_TP(IN := "DB1_SalidasExterioresDeMesa".Mesa[#Mesa].Bajar_TP_E1E3 AND #EnMovimiento_TP AND NOT #EstadoZona.Manual_CBx,   // "FB910_CNT_UHS"
                  R := NOT #EnMovimiento_TP,
                  PV := #V_TOut_TP,
                  BaseUnidades_ms := "CTE_BaseUnidades_1ms");
END_REGION

REGION Network 51: ERROR - TimeOut Bajar TP
   RUNG wire#powerrail
      Contact( #EstadoZona.Rearme_CBx )
      S_RS(operand := #EstadoVI.Err_TOut_Bajar_TP_E1_E3, s1 := #TOut_Bajar_TP.QU)
      S_Coil( #EstadoVI.Error_Mx )
   END_RUNG
   // the same network as SCL:
   IF #EstadoZona.Rearme_CBx THEN
       #EstadoVI.Err_TOut_Bajar_TP_E1_E3 := FALSE;   // RS flip-flop
   END_IF;
   IF #TOut_Bajar_TP.QU THEN #EstadoVI.Err_TOut_Bajar_TP_E1_E3 := TRUE; END_IF;
   IF #EstadoVI.Err_TOut_Bajar_TP_E1_E3 THEN #EstadoVI.Error_Mx := TRUE; END_IF;
END_REGION

REGION Network 52: TMP - ERROR - TimeOut Griper In / Out
   RUNG wire#powerrail
      #TOut_Gripper(IN := wire#w2, R := wire#w3, PV := #V_TOut_Gripper, BaseUnidades_ms := "CTE_BaseUnidades_1ms", QU =>, QD =>, CVU =>, CVD =>)
   END_RUNG
   RUNG wire#powerrail
      Contact( #MA_Gripper_Cerrar )
      wire#w1
      Contact( #EnMovimiento_Gripper )
      I_Contact( #EstadoZona.Manual_CBx )
   END_RUNG wire#w2
   RUNG wire#powerrail
      Contact( #MA_Gripper_Cerrar )
   END_RUNG wire#w1
   RUNG wire#powerrail
      I_Contact( #MA_Gripper_Cerrar )
      I_Contact( #MA_Gripper_Cerrar )
   END_RUNG wire#w3
   // the same network as SCL:
   #TOut_Gripper(IN := (#MA_Gripper_Cerrar OR #MA_Gripper_Cerrar) AND #EnMovimiento_Gripper AND NOT #EstadoZona.Manual_CBx,   // "FB910_CNT_UHS"
                 R := NOT #MA_Gripper_Cerrar AND NOT #MA_Gripper_Cerrar,
                 PV := #V_TOut_Gripper,
                 BaseUnidades_ms := "CTE_BaseUnidades_1ms");
END_REGION

REGION Network 53: ERROR - TimeOut Griper Abrir
   RUNG wire#powerrail
      Contact( #EstadoZona.Rearme_CBx )
      S_RS(operand := #EstadoVI.Err_Tout_Recoger_gripper, s1 := wire#w1)
      S_Coil( #EstadoVI.Error_Mx )
   END_RUNG
   RUNG wire#powerrail
      Contact( #TOut_Gripper.QU )
      Contact( #MA_Gripper_Abrir )
   END_RUNG wire#w1
   // the same network as SCL:
   IF #EstadoZona.Rearme_CBx THEN
       #EstadoVI.Err_Tout_Recoger_gripper := FALSE;   // RS flip-flop
   END_IF;
   IF #TOut_Gripper.QU AND #MA_Gripper_Abrir THEN #EstadoVI.Err_Tout_Recoger_gripper := TRUE; END_IF;
   IF #EstadoVI.Err_Tout_Recoger_gripper THEN #EstadoVI.Error_Mx := TRUE; END_IF;
END_REGION

REGION Network 54: ERROR - TimeOut Griper Cerrar
   RUNG wire#powerrail
      Contact( #EstadoZona.Rearme_CBx )
      S_RS(operand := #EstadoVI.Err_Tout_Sacar_gripper, s1 := wire#w1)
      S_Coil( #EstadoVI.Error_Mx )
   END_RUNG
   RUNG wire#powerrail
      Contact( #TOut_Gripper.QU )
      Contact( #MA_Gripper_Cerrar )
   END_RUNG wire#w1
   RUNG wire#powerrail
      Contact( #Mx_ET02 )
      I_Contact( #PhsMx )
      Contact( #Phs_en_Pinza )
      I_Contact( #Gripper_Close )
   END_RUNG wire#w1
   // the same network as SCL:
   IF #EstadoZona.Rearme_CBx THEN
       #EstadoVI.Err_Tout_Sacar_gripper := FALSE;   // RS flip-flop
   END_IF;
   IF (#TOut_Gripper.QU AND #MA_Gripper_Cerrar) OR (#Mx_ET02 AND NOT #PhsMx AND #Phs_en_Pinza AND NOT #Gripper_Close) THEN
       #EstadoVI.Err_Tout_Sacar_gripper := TRUE;
   END_IF;
   IF #EstadoVI.Err_Tout_Sacar_gripper THEN #EstadoVI.Error_Mx := TRUE; END_IF;
END_REGION

REGION Network 55: TMP - ERROR - TimeOut Cilindro Up / Down
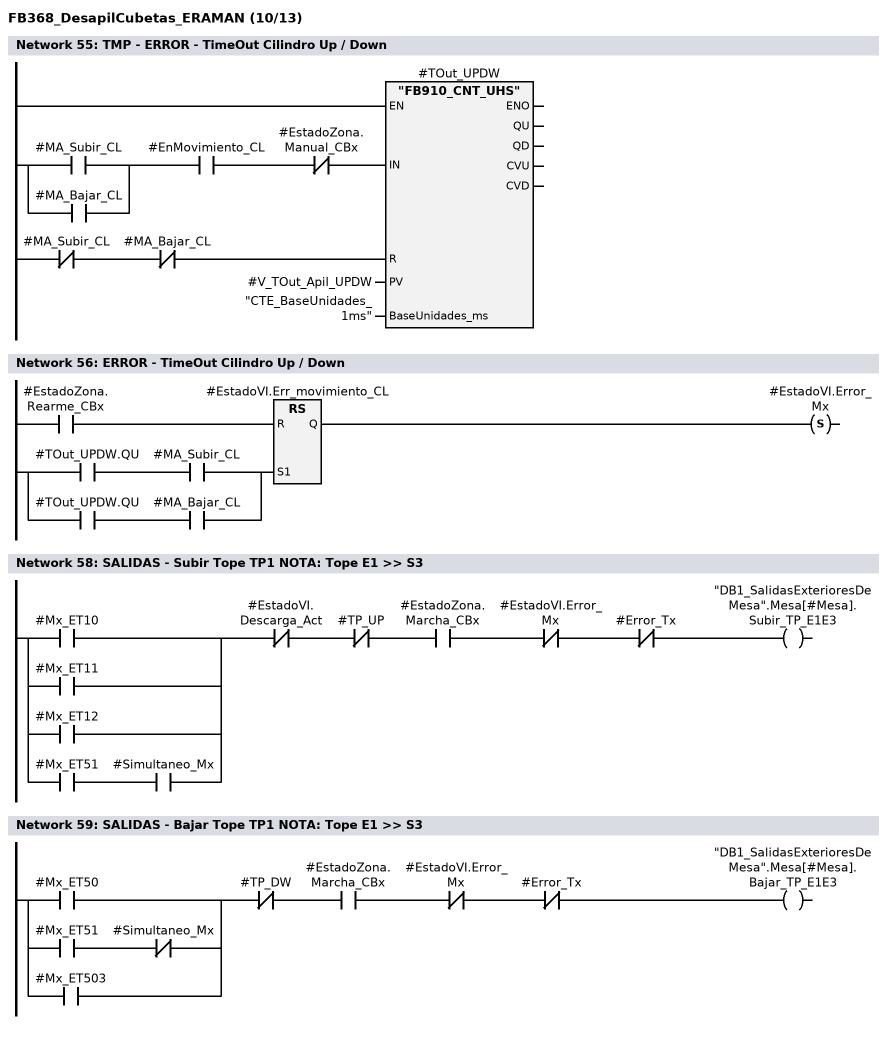
   RUNG wire#powerrail
      #TOut_UPDW(IN := wire#w2, R := wire#w3, PV := #V_TOut_Apil_UPDW, BaseUnidades_ms := "CTE_BaseUnidades_1ms", QU =>, QD =>, CVU =>, CVD =>)
   END_RUNG
   RUNG wire#powerrail
      Contact( #MA_Subir_CL )
      wire#w1
      Contact( #EnMovimiento_CL )
      I_Contact( #EstadoZona.Manual_CBx )
   END_RUNG wire#w2
   RUNG wire#powerrail
      Contact( #MA_Bajar_CL )
   END_RUNG wire#w1
   RUNG wire#powerrail
      I_Contact( #MA_Subir_CL )
      I_Contact( #MA_Bajar_CL )
   END_RUNG wire#w3
   // the same network as SCL:
   #TOut_UPDW(IN := (#MA_Subir_CL OR #MA_Bajar_CL) AND #EnMovimiento_CL AND NOT #EstadoZona.Manual_CBx,   // "FB910_CNT_UHS"
              R := NOT #MA_Subir_CL AND NOT #MA_Bajar_CL,
              PV := #V_TOut_Apil_UPDW,
              BaseUnidades_ms := "CTE_BaseUnidades_1ms");
END_REGION

REGION Network 56: ERROR - TimeOut Cilindro Up / Down
   RUNG wire#powerrail
      Contact( #EstadoZona.Rearme_CBx )
      S_RS(operand := #EstadoVI.Err_movimiento_CL, s1 := wire#w1)
      S_Coil( #EstadoVI.Error_Mx )
   END_RUNG
   RUNG wire#powerrail
      Contact( #TOut_UPDW.QU )
      Contact( #MA_Subir_CL )
   END_RUNG wire#w1
   RUNG wire#powerrail
      Contact( #TOut_UPDW.QU )
      Contact( #MA_Bajar_CL )
   END_RUNG wire#w1
   // the same network as SCL:
   IF #EstadoZona.Rearme_CBx THEN
       #EstadoVI.Err_movimiento_CL := FALSE;   // RS flip-flop
   END_IF;
   IF (#TOut_UPDW.QU AND #MA_Subir_CL) OR (#TOut_UPDW.QU AND #MA_Bajar_CL) THEN
       #EstadoVI.Err_movimiento_CL := TRUE;
   END_IF;
   IF #EstadoVI.Err_movimiento_CL THEN #EstadoVI.Error_Mx := TRUE; END_IF;
END_REGION

REGION Network 57: ----------------------SALIDAS -------------------------
END_REGION

REGION Network 58: SALIDAS - Subir Tope TP1 NOTA: Tope E1 >> S3
   RUNG wire#powerrail
      Contact( #Mx_ET10 )
      wire#w1
      I_Contact( #EstadoVI.Descarga_Act )
      I_Contact( #TP_UP )
      Contact( #EstadoZona.Marcha_CBx )
      I_Contact( #EstadoVI.Error_Mx )
      I_Contact( #Error_Tx )
      Coil( "DB1_SalidasExterioresDeMesa".Mesa[#Mesa].Subir_TP_E1E3 )
   END_RUNG
   RUNG wire#powerrail
      Contact( #Mx_ET11 )
   END_RUNG wire#w1
   RUNG wire#powerrail
      Contact( #Mx_ET12 )
   END_RUNG wire#w1
   RUNG wire#powerrail
      Contact( #Mx_ET51 )
      Contact( #Simultaneo_Mx )
   END_RUNG wire#w1
   // the same network as SCL:
   "DB1_SalidasExterioresDeMesa".Mesa[#Mesa].Subir_TP_E1E3 := (#Mx_ET10 OR #Mx_ET11 OR #Mx_ET12 OR (#Mx_ET51 AND #Simultaneo_Mx)) AND NOT #EstadoVI.Descarga_Act AND NOT #TP_UP AND #EstadoZona.Marcha_CBx AND NOT #EstadoVI.Error_Mx AND NOT #Error_Tx;
END_REGION

REGION Network 59: SALIDAS - Bajar Tope TP1 NOTA: Tope E1 >> S3
   RUNG wire#powerrail
      Contact( #Mx_ET50 )
      wire#w1
      I_Contact( #TP_DW )
      Contact( #EstadoZona.Marcha_CBx )
      I_Contact( #EstadoVI.Error_Mx )
      I_Contact( #Error_Tx )
      Coil( "DB1_SalidasExterioresDeMesa".Mesa[#Mesa].Bajar_TP_E1E3 )
   END_RUNG
   RUNG wire#powerrail
      Contact( #Mx_ET51 )
      I_Contact( #Simultaneo_Mx )
   END_RUNG wire#w1
   RUNG wire#powerrail
      Contact( #Mx_ET503 )
   END_RUNG wire#w1
   // the same network as SCL:
   "DB1_SalidasExterioresDeMesa".Mesa[#Mesa].Bajar_TP_E1E3 := (#Mx_ET50 OR (#Mx_ET51 AND NOT #Simultaneo_Mx) OR #Mx_ET503) AND NOT #TP_DW AND #EstadoZona.Marcha_CBx AND NOT #EstadoVI.Error_Mx AND NOT #Error_Tx;
END_REGION

REGION Network 60: SALIDAS - Avanzar E1E3
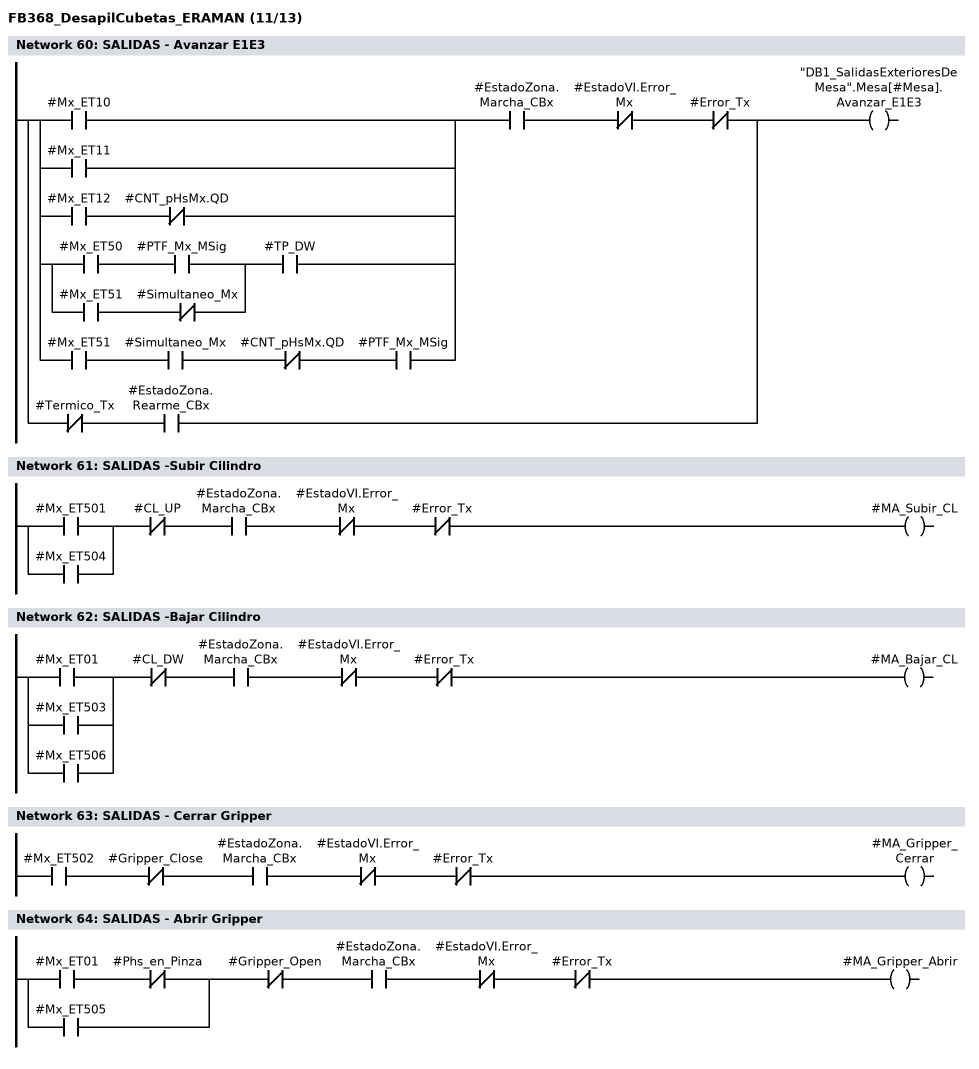
   RUNG wire#powerrail
      Contact( #Mx_ET10 )
      wire#w1
      Contact( #EstadoZona.Marcha_CBx )
      I_Contact( #EstadoVI.Error_Mx )
      I_Contact( #Error_Tx )
      wire#w3
      Coil( "DB1_SalidasExterioresDeMesa".Mesa[#Mesa].Avanzar_E1E3 )
   END_RUNG
   RUNG wire#powerrail
      Contact( #Mx_ET11 )
   END_RUNG wire#w1
   RUNG wire#powerrail
      Contact( #Mx_ET12 )
      I_Contact( #CNT_pHsMx.QD )
   END_RUNG wire#w1
   RUNG wire#powerrail
      Contact( #Mx_ET50 )
      Contact( #PTF_Mx_MSig )
      wire#w2
      Contact( #TP_DW )
   END_RUNG wire#w1
   RUNG wire#powerrail
      Contact( #Mx_ET51 )
      I_Contact( #Simultaneo_Mx )
   END_RUNG wire#w2
   RUNG wire#powerrail
      Contact( #Mx_ET51 )
      Contact( #Simultaneo_Mx )
      I_Contact( #CNT_pHsMx.QD )
      Contact( #PTF_Mx_MSig )
   END_RUNG wire#w1
   RUNG wire#powerrail
      I_Contact( #Termico_Tx )
      Contact( #EstadoZona.Rearme_CBx )
   END_RUNG wire#w3
   // the same network as SCL:
   "DB1_SalidasExterioresDeMesa".Mesa[#Mesa].Avanzar_E1E3 := ((#Mx_ET10 OR #Mx_ET11 OR (#Mx_ET12 AND NOT #CNT_pHsMx.QD) OR (((#Mx_ET50 AND #PTF_Mx_MSig) OR (#Mx_ET51 AND NOT #Simultaneo_Mx)) AND #TP_DW) OR (#Mx_ET51 AND #Simultaneo_Mx AND NOT #CNT_pHsMx.QD AND #PTF_Mx_MSig)) AND #EstadoZona.Marcha_CBx AND NOT #EstadoVI.Error_Mx AND NOT #Error_Tx) OR (NOT #Termico_Tx AND #EstadoZona.Rearme_CBx);
END_REGION

REGION Network 61: SALIDAS -Subir Cilindro
   RUNG wire#powerrail
      Contact( #Mx_ET501 )
      wire#w1
      I_Contact( #CL_UP )
      Contact( #EstadoZona.Marcha_CBx )
      I_Contact( #EstadoVI.Error_Mx )
      I_Contact( #Error_Tx )
      Coil( #MA_Subir_CL )
   END_RUNG
   RUNG wire#powerrail
      Contact( #Mx_ET504 )
   END_RUNG wire#w1
   // the same network as SCL:
   #MA_Subir_CL := (#Mx_ET501 OR #Mx_ET504) AND NOT #CL_UP AND #EstadoZona.Marcha_CBx AND NOT #EstadoVI.Error_Mx AND NOT #Error_Tx;
END_REGION

REGION Network 62: SALIDAS -Bajar Cilindro
   RUNG wire#powerrail
      Contact( #Mx_ET01 )
      wire#w1
      I_Contact( #CL_DW )
      Contact( #EstadoZona.Marcha_CBx )
      I_Contact( #EstadoVI.Error_Mx )
      I_Contact( #Error_Tx )
      Coil( #MA_Bajar_CL )
   END_RUNG
   RUNG wire#powerrail
      Contact( #Mx_ET503 )
   END_RUNG wire#w1
   RUNG wire#powerrail
      Contact( #Mx_ET506 )
   END_RUNG wire#w1
   // the same network as SCL:
   #MA_Bajar_CL := (#Mx_ET01 OR #Mx_ET503 OR #Mx_ET506) AND NOT #CL_DW AND #EstadoZona.Marcha_CBx AND NOT #EstadoVI.Error_Mx AND NOT #Error_Tx;
END_REGION

REGION Network 63: SALIDAS - Cerrar Gripper
   RUNG wire#powerrail
      Contact( #Mx_ET502 )
      I_Contact( #Gripper_Close )
      Contact( #EstadoZona.Marcha_CBx )
      I_Contact( #EstadoVI.Error_Mx )
      I_Contact( #Error_Tx )
      Coil( #MA_Gripper_Cerrar )
   END_RUNG
   // the same network as SCL:
   #MA_Gripper_Cerrar := #Mx_ET502 AND NOT #Gripper_Close AND #EstadoZona.Marcha_CBx AND NOT #EstadoVI.Error_Mx AND NOT #Error_Tx;
END_REGION

REGION Network 64: SALIDAS - Abrir Gripper
   RUNG wire#powerrail
      Contact( #Mx_ET01 )
      I_Contact( #Phs_en_Pinza )
      wire#w1
      I_Contact( #Gripper_Open )
      Contact( #EstadoZona.Marcha_CBx )
      I_Contact( #EstadoVI.Error_Mx )
      I_Contact( #Error_Tx )
      Coil( #MA_Gripper_Abrir )
   END_RUNG
   RUNG wire#powerrail
      Contact( #Mx_ET505 )
   END_RUNG wire#w1
   // the same network as SCL:
   #MA_Gripper_Abrir := ((#Mx_ET01 AND NOT #Phs_en_Pinza) OR #Mx_ET505) AND NOT #Gripper_Open AND #EstadoZona.Marcha_CBx AND NOT #EstadoVI.Error_Mx AND NOT #Error_Tx;
END_REGION

REGION Network 65: ---------------------- ESTADOS /ENTRADAS MESA -------------------------
END_REGION

REGION Network 66: ESTADOS DE LA MESA
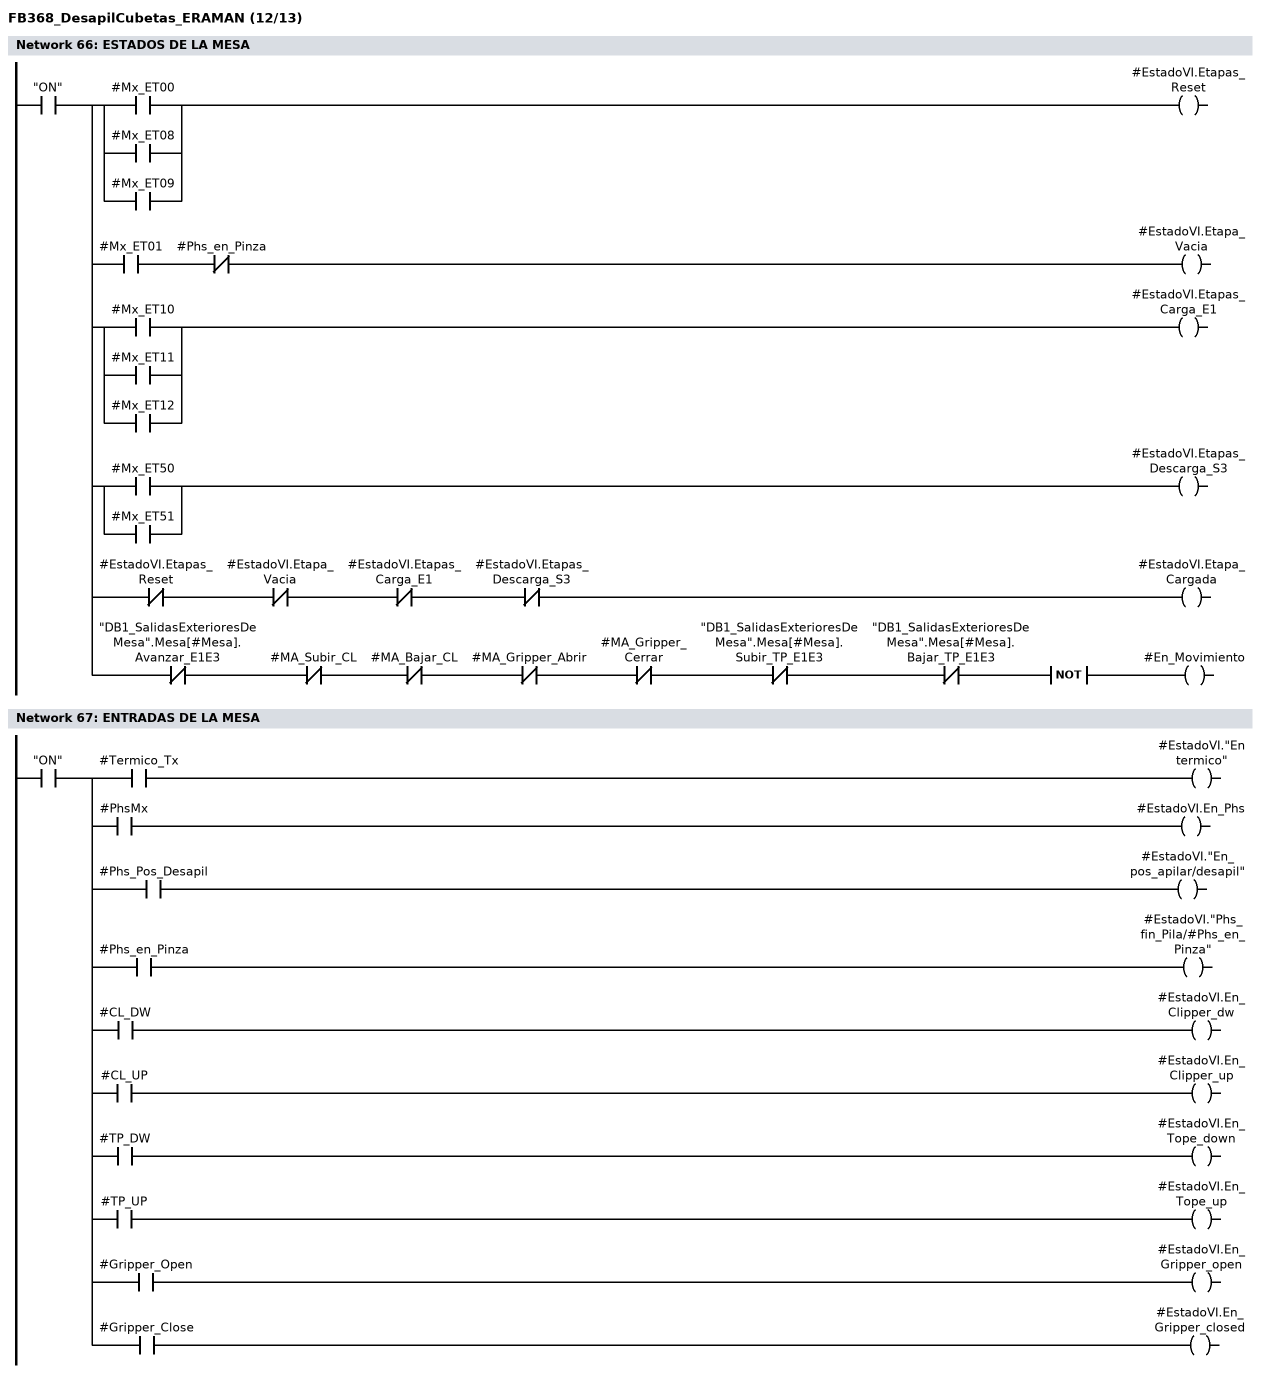
   RUNG wire#powerrail
      Contact( "ON" )
      wire#w1
      Contact( #Mx_ET00 )
      wire#w2
      Coil( #EstadoVI.Etapas_Reset )
   END_RUNG
   RUNG wire#w1
      Contact( #Mx_ET08 )
   END_RUNG wire#w2
   RUNG wire#w1
      Contact( #Mx_ET09 )
   END_RUNG wire#w2
   RUNG wire#w1
      Contact( #Mx_ET01 )
      I_Contact( #Phs_en_Pinza )
      Coil( #EstadoVI.Etapa_Vacia )
   END_RUNG
   RUNG wire#w1
      Contact( #Mx_ET10 )
      wire#w3
      Coil( #EstadoVI.Etapas_Carga_E1 )
   END_RUNG
   RUNG wire#w1
      Contact( #Mx_ET11 )
   END_RUNG wire#w3
   RUNG wire#w1
      Contact( #Mx_ET12 )
   END_RUNG wire#w3
   RUNG wire#w1
      Contact( #Mx_ET50 )
      wire#w4
      Coil( #EstadoVI.Etapas_Descarga_S3 )
   END_RUNG
   RUNG wire#w1
      Contact( #Mx_ET51 )
   END_RUNG wire#w4
   RUNG wire#w1
      I_Contact( #EstadoVI.Etapas_Reset )
      I_Contact( #EstadoVI.Etapa_Vacia )
      I_Contact( #EstadoVI.Etapas_Carga_E1 )
      I_Contact( #EstadoVI.Etapas_Descarga_S3 )
      Coil( #EstadoVI.Etapa_Cargada )
   END_RUNG
   RUNG wire#w1
      I_Contact( "DB1_SalidasExterioresDeMesa".Mesa[#Mesa].Avanzar_E1E3 )
      I_Contact( #MA_Subir_CL )
      I_Contact( #MA_Bajar_CL )
      I_Contact( #MA_Gripper_Abrir )
      I_Contact( #MA_Gripper_Cerrar )
      I_Contact( "DB1_SalidasExterioresDeMesa".Mesa[#Mesa].Subir_TP_E1E3 )
      I_Contact( "DB1_SalidasExterioresDeMesa".Mesa[#Mesa].Bajar_TP_E1E3 )
      Not()
      Coil( #En_Movimiento )
   END_RUNG
   // the same network as SCL:
   #EstadoVI.Etapas_Reset := "ON" AND (#Mx_ET00 OR #Mx_ET08 OR #Mx_ET09);
   #EstadoVI.Etapa_Vacia := "ON" AND #Mx_ET01 AND NOT #Phs_en_Pinza;
   #EstadoVI.Etapas_Carga_E1 := "ON" AND (#Mx_ET10 OR #Mx_ET11 OR #Mx_ET12);
   #EstadoVI.Etapas_Descarga_S3 := "ON" AND (#Mx_ET50 OR #Mx_ET51);
   #EstadoVI.Etapa_Cargada := "ON" AND NOT #EstadoVI.Etapas_Reset AND NOT #EstadoVI.Etapa_Vacia AND NOT #EstadoVI.Etapas_Carga_E1 AND NOT #EstadoVI.Etapas_Descarga_S3;
   #En_Movimiento := NOT ("ON" AND NOT "DB1_SalidasExterioresDeMesa".Mesa[#Mesa].Avanzar_E1E3 AND NOT #MA_Subir_CL AND NOT #MA_Bajar_CL AND NOT #MA_Gripper_Abrir AND NOT #MA_Gripper_Cerrar AND NOT "DB1_SalidasExterioresDeMesa".Mesa[#Mesa].Subir_TP_E1E3 AND NOT "DB1_SalidasExterioresDeMesa".Mesa[#Mesa].Bajar_TP_E1E3);
END_REGION

REGION Network 67: ENTRADAS DE LA MESA
   RUNG wire#powerrail
      Contact( "ON" )
      wire#w1
      Contact( #Termico_Tx )
      Coil( #EstadoVI."En termico" )
   END_RUNG
   RUNG wire#w1
      Contact( #PhsMx )
      Coil( #EstadoVI.En_Phs )
   END_RUNG
   RUNG wire#w1
      Contact( #Phs_Pos_Desapil )
      Coil( #EstadoVI."En_pos_apilar/desapil" )
   END_RUNG
   RUNG wire#w1
      Contact( #Phs_en_Pinza )
      Coil( #EstadoVI."Phs_fin_Pila/#Phs_en_Pinza" )
   END_RUNG
   RUNG wire#w1
      Contact( #CL_DW )
      Coil( #EstadoVI.En_Clipper_dw )
   END_RUNG
   RUNG wire#w1
      Contact( #CL_UP )
      Coil( #EstadoVI.En_Clipper_up )
   END_RUNG
   RUNG wire#w1
      Contact( #TP_DW )
      Coil( #EstadoVI.En_Tope_down )
   END_RUNG
   RUNG wire#w1
      Contact( #TP_UP )
      Coil( #EstadoVI.En_Tope_up )
   END_RUNG
   RUNG wire#w1
      Contact( #Gripper_Open )
      Coil( #EstadoVI.En_Gripper_open )
   END_RUNG
   RUNG wire#w1
      Contact( #Gripper_Close )
      Coil( #EstadoVI.En_Gripper_closed )
   END_RUNG
   // the same network as SCL:
   #EstadoVI."En termico" := "ON" AND #Termico_Tx;
   #EstadoVI.En_Phs := "ON" AND #PhsMx;
   #EstadoVI."En_pos_apilar/desapil" := "ON" AND #Phs_Pos_Desapil;
   #EstadoVI."Phs_fin_Pila/#Phs_en_Pinza" := "ON" AND #Phs_en_Pinza;
   #EstadoVI.En_Clipper_dw := "ON" AND #CL_DW;
   #EstadoVI.En_Clipper_up := "ON" AND #CL_UP;
   #EstadoVI.En_Tope_down := "ON" AND #TP_DW;
   #EstadoVI.En_Tope_up := "ON" AND #TP_UP;
   #EstadoVI.En_Gripper_open := "ON" AND #Gripper_Open;
   #EstadoVI.En_Gripper_closed := "ON" AND #Gripper_Close;
END_REGION

REGION Network 68: SALIDAS DE LA MESA
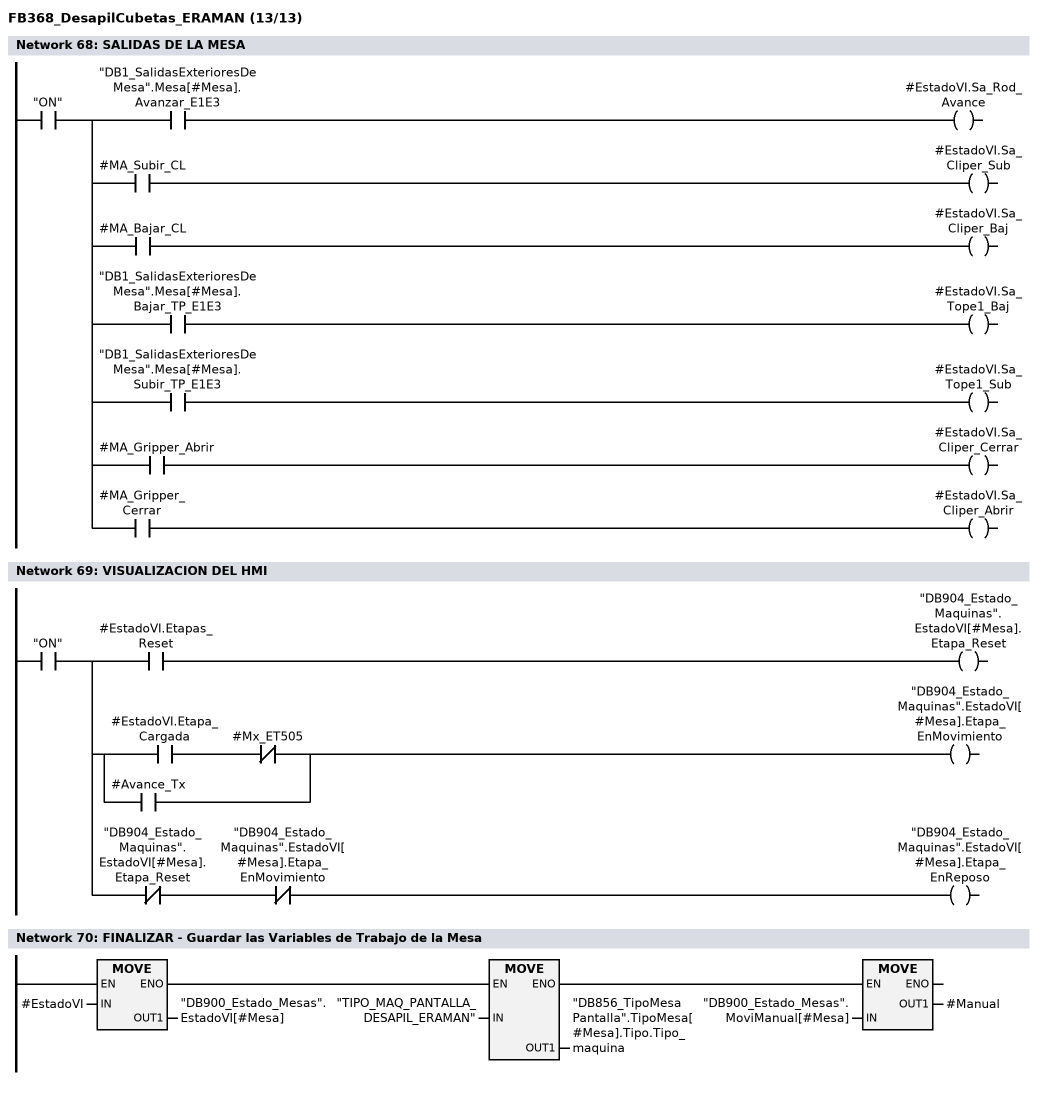
   RUNG wire#powerrail
      Contact( "ON" )
      wire#w1
      Contact( "DB1_SalidasExterioresDeMesa".Mesa[#Mesa].Avanzar_E1E3 )
      Coil( #EstadoVI.Sa_Rod_Avance )
   END_RUNG
   RUNG wire#w1
      Contact( #MA_Subir_CL )
      Coil( #EstadoVI.Sa_Cliper_Sub )
   END_RUNG
   RUNG wire#w1
      Contact( #MA_Bajar_CL )
      Coil( #EstadoVI.Sa_Cliper_Baj )
   END_RUNG
   RUNG wire#w1
      Contact( "DB1_SalidasExterioresDeMesa".Mesa[#Mesa].Bajar_TP_E1E3 )
      Coil( #EstadoVI.Sa_Tope1_Baj )
   END_RUNG
   RUNG wire#w1
      Contact( "DB1_SalidasExterioresDeMesa".Mesa[#Mesa].Subir_TP_E1E3 )
      Coil( #EstadoVI.Sa_Tope1_Sub )
   END_RUNG
   RUNG wire#w1
      Contact( #MA_Gripper_Abrir )
      Coil( #EstadoVI.Sa_Cliper_Cerrar )
   END_RUNG
   RUNG wire#w1
      Contact( #MA_Gripper_Cerrar )
      Coil( #EstadoVI.Sa_Cliper_Abrir )
   END_RUNG
   // the same network as SCL:
   #EstadoVI.Sa_Rod_Avance := "ON" AND "DB1_SalidasExterioresDeMesa".Mesa[#Mesa].Avanzar_E1E3;
   #EstadoVI.Sa_Cliper_Sub := "ON" AND #MA_Subir_CL;
   #EstadoVI.Sa_Cliper_Baj := "ON" AND #MA_Bajar_CL;
   #EstadoVI.Sa_Tope1_Baj := "ON" AND "DB1_SalidasExterioresDeMesa".Mesa[#Mesa].Bajar_TP_E1E3;
   #EstadoVI.Sa_Tope1_Sub := "ON" AND "DB1_SalidasExterioresDeMesa".Mesa[#Mesa].Subir_TP_E1E3;
   #EstadoVI.Sa_Cliper_Cerrar := "ON" AND #MA_Gripper_Abrir;
   #EstadoVI.Sa_Cliper_Abrir := "ON" AND #MA_Gripper_Cerrar;
END_REGION

REGION Network 69: VISUALIZACION DEL HMI
   RUNG wire#powerrail
      Contact( "ON" )
      wire#w1
      Contact( #EstadoVI.Etapas_Reset )
      Coil( "DB904_Estado_Maquinas".EstadoVI[#Mesa].Etapa_Reset )
   END_RUNG
   RUNG wire#w1
      Contact( #EstadoVI.Etapa_Cargada )
      I_Contact( #Mx_ET505 )
      wire#w2
      Coil( "DB904_Estado_Maquinas".EstadoVI[#Mesa].Etapa_EnMovimiento )
   END_RUNG
   RUNG wire#w1
      Contact( #Avance_Tx )
   END_RUNG wire#w2
   RUNG wire#w1
      I_Contact( "DB904_Estado_Maquinas".EstadoVI[#Mesa].Etapa_Reset )
      I_Contact( "DB904_Estado_Maquinas".EstadoVI[#Mesa].Etapa_EnMovimiento )
      Coil( "DB904_Estado_Maquinas".EstadoVI[#Mesa].Etapa_EnReposo )
   END_RUNG
   // the same network as SCL:
   "DB904_Estado_Maquinas".EstadoVI[#Mesa].Etapa_Reset := "ON" AND #EstadoVI.Etapas_Reset;
   "DB904_Estado_Maquinas".EstadoVI[#Mesa].Etapa_EnMovimiento := "ON" AND ((#EstadoVI.Etapa_Cargada AND NOT #Mx_ET505) OR #Avance_Tx);
   "DB904_Estado_Maquinas".EstadoVI[#Mesa].Etapa_EnReposo := "ON" AND NOT "DB904_Estado_Maquinas".EstadoVI[#Mesa].Etapa_Reset AND NOT "DB904_Estado_Maquinas".EstadoVI[#Mesa].Etapa_EnMovimiento;
END_REGION

REGION Network 70: FINALIZAR - Guardar las Variables de Trabajo de la Mesa
   RUNG wire#powerrail
      Move(in := #EstadoVI, out1 => "DB900_Estado_Mesas".EstadoVI[#Mesa])
      Move(in := "TIPO_MAQ_PANTALLA_DESAPIL_ERAMAN", out1 => "DB856_TipoMesaPantalla".TipoMesa[#Mesa].Tipo.Tipo_maquina)
      Move(in := "DB900_Estado_Mesas".MoviManual[#Mesa], out1 => #Manual)
   END_RUNG
   // the same network as SCL:
   "DB900_Estado_Mesas".EstadoVI[#Mesa] := #EstadoVI;
   "DB856_TipoMesaPantalla".TipoMesa[#Mesa].Tipo.Tipo_maquina := "TIPO_MAQ_PANTALLA_DESAPIL_ERAMAN";
   #Manual := "DB900_Estado_Mesas".MoviManual[#Mesa];
END_REGION
END_FUNCTION_BLOCK
